C09157=1149.476,8.134,-48.383,179.808,6.183,149.173
C09158=1149.470,8.383,-48.397,179.810,6.184,149.172
C09159=1149.465,8.633,-48.412,179.813,6.186,149.172
C09160=1149.460,8.883,-48.425,179.816,6.186,149.171
C09161=1149.455,9.132,-48.438,179.818,6.187,149.171
C09162=1149.450,9.382,-48.452,179.821,6.187,149.170
C09163=1149.444,9.631,-48.466,179.823,6.188,149.169
C09164=1149.440,9.881,-48.480,179.826,6.189,149.169
C09165=1149.435,10.131,-48.493,179.828,6.190,149.168
C09166=1149.429,10.380,-48.507,179.830,6.191,149.168
C09167=1149.424,10.630,-48.521,179.833,6.191,149.167
C09168=1149.419,10.879,-48.534,179.835,6.192,149.167
C09169=1149.414,11.129,-48.548,179.838,6.193,149.166
C09170=1149.409,11.379,-48.562,179.841,6.194,149.165
C09171=1149.403,11.628,-48.576,179.843,6.195,149.165
C09172=1149.399,11.877,-48.589,179.845,6.196,149.164
C09173=1149.394,12.126,-48.603,179.849,6.197,149.164
C09174=1149.388,12.377,-48.617,179.851,6.198,149.163
C09175=1149.383,12.627,-48.631,179.853,6.198,149.163
C09176=1149.378,12.876,-48.645,179.856,6.199,149.162
C09177=1149.373,13.126,-48.658,179.858,6.201,149.162
C09178=1149.368,13.375,-48.672,179.861,6.201,149.161
C09179=1149.363,13.624,-48.686,179.863,6.202,149.160
C09180=1149.358,13.874,-48.700,179.866,6.202,149.160
C09181=1149.352,14.124,-48.714,179.868,6.203,149.159
C09182=1149.347,14.373,-48.728,179.871,6.204,149.159
C09183=1149.343,14.623,-48.742,179.873,6.205,149.158
C09184=1149.338,14.872,-48.756,179.876,6.206,149.157
C09185=1149.332,15.121,-48.770,179.878,6.206,149.157
C09186=1149.327,15.372,-48.783,179.882,6.208,149.156
C09187=1149.322,15.621,-48.798,179.884,6.208,149.156
C09188=1149.316,15.870,-48.812,179.886,6.209,149.155
C09189=1149.311,16.120,-48.826,179.889,6.210,149.155
C09190=1149.307,16.370,-48.840,179.891,6.211,149.154
C09191=1149.302,16.619,-48.853,179.894,6.212,149.154
C09192=1149.297,16.868,-48.868,179.896,6.213,149.153
C09193=1149.291,17.119,-48.881,179.899,6.213,149.152
C09194=1149.287,17.368,-48.896,179.902,6.215,149.152
C09195=1149.281,17.617,-48.909,179.904,6.215,149.151
C09196=1149.276,17.867,-48.924,179.906,6.216,149.151
C09197=1149.271,18.117,-48.938,179.909,6.218,149.150
C09198=1149.266,18.367,-48.952,179.912,6.218,149.150
C09199=1149.261,18.616,-48.966,179.914,6.219,149.149
C09200=1149.256,18.865,-48.980,179.917,6.219,149.149
C09201=1149.251,19.115,-48.995,179.919,6.221,149.148
C09202=1149.246,19.364,-49.008,179.922,6.221,149.147
C09203=1149.241,19.613,-49.022,179.924,6.222,149.147
C09204=1149.236,19.863,-49.037,179.927,6.223,149.146
C09205=1149.231,20.113,-49.051,179.930,6.224,149.146
C09206=1149.226,20.362,-49.065,179.932,6.225,149.145
C09207=1149.220,20.611,-49.079,179.934,6.226,149.145
C09208=1149.215,20.861,-49.093,179.937,6.227,149.144
C09209=1149.211,21.111,-49.108,179.940,6.228,149.144
C09210=1149.206,21.361,-49.122,179.942,6.229,149.143
C09211=1149.200,21.610,-49.136,179.945,6.229,149.142
C09212=1149.195,21.859,-49.150,179.947,6.231,149.142
C09213=1149.190,22.109,-49.164,179.950,6.231,149.141
C09214=1149.185,22.359,-49.179,179.952,6.232,149.141
C09215=1149.179,22.609,-49.194,179.955,6.233,149.140
C09216=1149.174,22.858,-49.207,179.958,6.234,149.140
C09217=1149.169,23.107,-49.222,179.960,6.235,149.139
C09218=1149.164,23.357,-49.236,179.962,6.235,149.139
C09219=1149.159,23.607,-49.250,179.965,6.237,149.138
C09220=1149.154,23.857,-49.265,179.968,6.237,149.137
C09221=1149.149,24.106,-49.280,179.970,6.238,149.137
C09222=1149.144,24.355,-49.293,179.973,6.239,149.136
C09223=1149.139,24.604,-49.308,179.975,6.240,149.136
C09224=1149.134,24.854,-49.322,179.978,6.241,149.135
C09225=1149.129,25.104,-49.336,179.981,6.242,149.135
C09226=1149.124,25.354,-49.351,179.983,6.243,149.134
C09227=1149.119,25.603,-49.366,179.986,6.244,149.134
C09228=1149.113,25.852,-49.380,179.988,6.245,149.133
C09229=1149.108,26.102,-49.394,179.991,6.246,149.132
C09230=1149.103,26.351,-49.409,179.993,6.247,149.132
C09231=1149.098,26.601,-49.423,179.996,6.247,149.131
C09232=1149.094,26.850,-49.438,179.999,6.249,149.131
C09233=1149.089,27.100,-49.452,-179.999,6.249,149.130
C09234=1149.083,27.369,-49.468,-179.996,6.251,149.130
C09235=1149.077,27.638,-49.483,-179.993,6.251,149.129
C09236=1149.072,27.907,-49.499,-179.991,6.253,149.129
C09237=1149.067,28.175,-49.515,-179.988,6.253,149.128
C09238=1149.061,28.425,-49.529,-179.986,6.254,149.127
C09239=1149.056,28.675,-49.544,-179.982,6.255,149.127
C09240=1149.051,28.924,-49.559,-179.980,6.256,149.126
C09241=1149.046,29.174,-49.573,-179.978,6.257,149.126
C09242=1149.041,29.424,-49.587,-179.975,6.258,149.125
C09243=1149.036,29.673,-49.603,-179.972,6.259,149.125
C09244=1149.031,29.923,-49.617,-179.970,6.260,149.124
C09245=1149.026,30.172,-49.631,-179.967,6.261,149.124
C09246=1149.021,30.421,-49.646,-179.965,6.262,149.123
C09247=1149.016,30.671,-49.661,-179.962,6.263,149.122
C09248=1149.011,30.921,-49.676,-179.959,6.264,149.122
C09249=1149.006,31.170,-49.690,-179.957,6.265,149.121
C09250=1149.001,31.419,-49.704,-179.954,6.266,149.121
C09251=1148.995,31.669,-49.720,-179.952,6.267,149.120
C09252=1148.990,31.918,-49.734,-179.950,6.268,149.120
C09253=1148.986,32.167,-49.749,-179.946,6.269,149.119
C09254=1148.981,32.417,-49.764,-179.944,6.270,149.119
C09255=1148.975,32.667,-49.778,-179.942,6.270,149.118
C09256=1148.970,32.916,-49.793,-179.939,6.272,149.118
C09257=1148.965,33.166,-49.808,-179.936,6.272,149.117
C09258=1148.960,33.415,-49.823,-179.934,6.273,149.116
C09259=1148.955,33.665,-49.838,-179.931,6.275,149.116
C09260=1148.950,33.914,-49.853,-179.929,6.275,149.115
C09261=1148.945,34.164,-49.867,-179.926,6.277,149.115
C09262=1148.940,34.413,-49.882,-179.923,6.277,149.114
C09263=1148.935,34.663,-49.897,-179.921,6.278,149.114
C09264=1148.930,34.912,-49.912,-179.918,6.279,149.113
C09265=1148.925,35.162,-49.927,-179.916,6.280,149.113
C09266=1148.920,35.411,-49.942,-179.913,6.281,149.112
C09267=1148.914,35.661,-49.956,-179.910,6.282,149.111
C09268=1148.910,35.910,-49.971,-179.908,6.283,149.111
C09269=1148.904,36.160,-49.987,-179.905,6.284,149.110
C09270=1148.899,36.409,-50.001,-179.903,6.285,149.110
C09271=1148.895,36.659,-50.016,-179.900,6.286,149.109
C09272=1148.890,36.909,-50.031,-179.897,6.287,149.109
C09273=1148.885,37.158,-50.046,-179.895,6.288,149.108
C09274=1148.880,37.408,-50.062,-179.892,6.289,149.108
C09275=1148.875,37.658,-50.076,-179.890,6.290,149.107
C09276=1148.869,37.907,-50.092,-179.887,6.291,149.106
C09277=1148.864,38.157,-50.106,-179.884,6.292,149.106
C09278=1148.860,38.406,-50.121,-179.882,6.293,149.106
C09279=1148.854,38.655,-50.137,-179.879,6.294,149.105
C09280=1148.849,38.905,-50.151,-179.877,6.295,149.104
C09281=1148.844,39.154,-50.167,-179.874,6.296,149.104
C09282=1148.839,39.403,-50.182,-179.871,6.297,149.103
C09283=1148.834,39.653,-50.197,-179.869,6.298,149.103
C09284=1148.829,39.902,-50.212,-179.866,6.299,149.102
C09285=1148.823,40.152,-50.227,-179.864,6.300,149.102
C09286=1148.819,40.402,-50.242,-179.861,6.301,149.101
C09287=1148.814,40.652,-50.257,-179.858,6.302,149.101
C09288=1148.809,40.901,-50.272,-179.856,6.303,149.100
C09289=1148.804,41.150,-50.288,-179.853,6.305,149.100
C09290=1148.799,41.399,-50.303,-179.851,6.305,149.099
C09291=1148.793,41.649,-50.318,-179.848,6.306,149.098
C09292=1148.789,41.898,-50.333,-179.845,6.308,149.098
C09293=1148.783,42.148,-50.348,-179.843,6.308,149.097
C09294=1148.779,42.398,-50.364,-179.840,6.310,149.097
C09295=1148.774,42.647,-50.379,-179.838,6.310,149.096
C09296=1148.768,42.897,-50.394,-179.835,6.312,149.096
C09297=1148.764,43.146,-50.409,-179.832,6.313,149.095
C09298=1148.758,43.395,-50.425,-179.830,6.313,149.095
C09299=1148.754,43.645,-50.440,-179.827,6.315,149.094
C09300=1148.749,43.895,-50.456,-179.825,6.316,149.094
C09301=1148.743,44.144,-50.471,-179.822,6.317,149.093
C09302=1148.739,44.393,-50.486,-179.819,6.318,149.093
C09303=1148.733,44.643,-50.501,-179.816,6.319,149.092
C09304=1148.728,44.892,-50.516,-179.814,6.320,149.091
C09305=1148.723,45.142,-50.532,-179.811,6.321,149.091
C09306=1148.718,45.392,-50.548,-179.809,6.322,149.090
C09307=1148.714,45.641,-50.563,-179.806,6.323,149.090
C09308=1148.708,45.890,-50.578,-179.803,6.324,149.089
C09309=1148.703,46.140,-50.594,-179.801,6.325,149.089
C09310=1148.698,46.389,-50.609,-179.798,6.326,149.088
C09311=1148.693,46.639,-50.625,-179.796,6.327,149.088
C09312=1148.688,46.888,-50.640,-179.793,6.329,149.087
C09313=1148.683,47.137,-50.655,-179.790,6.329,149.087
C09314=1148.678,47.387,-50.671,-179.788,6.331,149.086
C09315=1148.673,47.637,-50.687,-179.785,6.332,149.086
C09316=1148.668,47.886,-50.702,-179.782,6.333,149.085
C09317=1148.663,48.135,-50.718,-179.780,6.334,149.085
C09318=1148.658,48.385,-50.733,-179.777,6.334,149.084
C09319=1148.654,48.635,-50.748,-179.775,6.336,149.083
C09320=1148.648,48.884,-50.764,-179.772,6.337,149.083
C09321=1148.643,49.133,-50.780,-179.769,6.338,149.082
C09322=1148.637,49.383,-50.795,-179.767,6.339,149.082
C09323=1148.633,49.633,-50.811,-179.764,6.340,149.081
C09324=1148.628,49.882,-50.826,-179.762,6.341,149.081
C09325=1148.623,50.131,-50.842,-179.759,6.343,149.080
C09326=1148.618,50.381,-50.858,-179.756,6.343,149.080
C09327=1148.614,50.630,-50.873,-179.754,6.345,149.079
C09328=1148.608,50.879,-50.889,-179.751,6.346,149.079
C09329=1148.603,51.129,-50.905,-179.748,6.347,149.078
C09330=1148.598,51.379,-50.921,-179.746,6.348,149.078
C09331=1148.593,51.628,-50.936,-179.743,6.349,149.077
C09332=1148.588,51.877,-50.951,-179.741,6.350,149.077
C09333=1148.583,52.127,-50.968,-179.738,6.351,149.076
C09334=1148.578,52.376,-50.983,-179.735,6.352,149.075
C09335=1148.573,52.626,-50.999,-179.732,6.354,149.075
C09336=1148.568,52.876,-51.015,-179.730,6.354,149.074
C09337=1148.563,53.125,-51.030,-179.727,6.356,149.074
C09338=1148.558,53.393,-51.047,-179.725,6.357,149.073
C09339=1148.552,53.662,-51.064,-179.722,6.358,149.073
C09340=1148.547,53.931,-51.081,-179.718,6.359,149.072
C09341=1148.542,54.199,-51.098,-179.716,6.360,149.072
C09342=1148.536,54.449,-51.114,-179.713,6.361,149.071
C09343=1148.531,54.698,-51.130,-179.711,6.362,149.071
C09344=1148.526,54.948,-51.146,-179.708,6.364,149.070
C09345=1148.521,55.197,-51.162,-179.705,6.365,149.069
C09346=1148.517,55.446,-51.178,-179.703,6.366,149.069
C09347=1148.512,55.696,-51.193,-179.700,6.368,149.069
C09348=1148.506,55.945,-51.209,-179.697,6.368,149.068
C09349=1148.502,56.195,-51.226,-179.695,6.370,149.068
C09350=1148.497,56.444,-51.241,-179.692,6.370,149.067
C09351=1148.491,56.693,-51.257,-179.689,6.372,149.066
C09352=1148.487,56.943,-51.274,-179.687,6.373,149.066
C09353=1148.481,57.192,-51.289,-179.684,6.374,149.065
C09354=1148.477,57.442,-51.305,-179.682,6.375,149.065
C09355=1148.471,57.691,-51.321,-179.679,6.376,149.064
C09356=1148.466,57.941,-51.337,-179.676,6.377,149.064
C09357=1148.462,58.190,-51.354,-179.674,6.379,149.063
C09358=1148.456,58.439,-51.369,-179.671,6.379,149.063
C09359=1148.451,58.690,-51.385,-179.668,6.381,149.062
C09360=1148.446,58.938,-51.402,-179.666,6.382,149.062
C09361=1148.442,59.188,-51.417,-179.663,6.383,149.061
C09362=1148.436,59.437,-51.434,-179.660,6.384,149.061
C09363=1148.432,59.687,-51.450,-179.658,6.385,149.060
C09364=1148.427,59.936,-51.466,-179.655,6.387,149.060
C09365=1148.421,60.186,-51.482,-179.652,6.387,149.059
C09366=1148.417,60.435,-51.498,-179.650,6.389,149.059
C09367=1148.411,60.684,-51.514,-179.647,6.390,149.058
C09368=1148.407,60.934,-51.531,-179.644,6.391,149.058
C09369=1148.401,61.183,-51.546,-179.642,6.392,149.057
C09370=1148.397,61.433,-51.563,-179.639,6.393,149.056
C09371=1148.392,61.682,-51.578,-179.637,6.394,149.056
C09372=1148.387,61.932,-51.595,-179.634,6.396,149.056
C09373=1148.382,62.181,-51.611,-179.631,6.397,149.055
C09374=1148.377,62.431,-51.627,-179.629,6.398,149.055
C09375=1148.372,62.679,-51.644,-179.625,6.399,149.054
C09376=1148.367,62.930,-51.660,-179.623,6.400,149.053
C09377=1148.362,63.179,-51.676,-179.621,6.402,149.053
C09378=1148.357,63.429,-51.692,-179.618,6.402,149.052
C09379=1148.352,63.677,-51.709,-179.615,6.404,149.052
C09380=1148.347,63.927,-51.725,-179.612,6.406,149.051
C09381=1148.342,64.176,-51.741,-179.610,6.406,149.051
C09382=1148.337,64.426,-51.758,-179.607,6.408,149.050
C09383=1148.332,64.675,-51.774,-179.605,6.409,149.050
C09384=1148.327,64.925,-51.790,-179.602,6.410,149.049
C09385=1148.322,65.174,-51.807,-179.600,6.411,149.049
C09386=1148.317,65.423,-51.823,-179.597,6.412,149.048
C09387=1148.312,65.673,-51.839,-179.594,6.414,149.048
C09388=1148.307,65.922,-51.856,-179.591,6.415,149.047
C09389=1148.303,66.172,-51.872,-179.589,6.416,149.047
C09390=1148.297,66.421,-51.889,-179.586,6.417,149.046
C09391=1148.292,66.671,-51.905,-179.583,6.418,149.046
C09392=1148.288,66.920,-51.922,-179.581,6.420,149.045
C09393=1148.283,67.169,-51.938,-179.578,6.421,149.045
C09394=1148.278,67.419,-51.955,-179.575,6.422,149.044
C09395=1148.272,67.668,-51.971,-179.573,6.423,149.044
C09396=1148.268,67.918,-51.988,-179.570,6.424,149.043
C09397=1148.263,68.167,-52.004,-179.567,6.426,149.043
C09398=1148.258,68.416,-52.021,-179.565,6.427,149.042
C09399=1148.253,68.666,-52.038,-179.562,6.428,149.042
C09400=1148.247,68.915,-52.054,-179.559,6.429,149.041
C09401=1148.243,69.165,-52.070,-179.557,6.431,149.041
C09402=1148.238,69.414,-52.087,-179.554,6.432,149.040
C09403=1148.233,69.663,-52.104,-179.551,6.433,149.040
C09404=1148.228,69.913,-52.120,-179.549,6.435,149.039
C09405=1148.224,70.162,-52.137,-179.545,6.436,149.039
C09406=1148.218,70.411,-52.154,-179.543,6.437,149.038
C09407=1148.213,70.661,-52.171,-179.540,6.438,149.038
C09408=1148.208,70.910,-52.186,-179.538,6.439,149.037
C09409=1148.203,71.160,-52.204,-179.535,6.441,149.037
C09410=1148.198,71.410,-52.220,-179.532,6.442,149.036
C09411=1148.193,71.658,-52.237,-179.530,6.443,149.036
C09412=1148.188,71.908,-52.254,-179.527,6.444,149.035
C09413=1148.184,72.158,-52.270,-179.524,6.446,149.035
C09414=1148.178,72.406,-52.287,-179.522,6.446,149.034
C09415=1148.173,72.656,-52.304,-179.519,6.448,149.034
C09416=1148.169,72.906,-52.321,-179.517,6.449,149.033
C09417=1148.164,73.155,-52.337,-179.514,6.450,149.032
C09418=1148.158,73.404,-52.354,-179.511,6.452,149.032
C09419=1148.154,73.654,-52.371,-179.509,6.453,149.032
C09420=1148.149,73.904,-52.388,-179.506,6.455,149.031
C09421=1148.144,74.152,-52.405,-179.503,6.456,149.031
C09422=1148.139,74.402,-52.421,-179.501,6.457,149.030
C09423=1148.134,74.652,-52.438,-179.498,6.458,149.030
C09424=1148.130,74.901,-52.455,-179.495,6.460,149.029
C09425=1148.124,75.150,-52.473,-179.492,6.460,149.029
C09426=1148.120,75.399,-52.489,-179.490,6.462,149.028
C09427=1148.114,75.649,-52.507,-179.486,6.463,149.027
C09428=1148.110,75.898,-52.523,-179.484,6.464,149.027
C09429=1148.104,76.147,-52.540,-179.482,6.466,149.027
C09430=1148.100,76.397,-52.557,-179.478,6.467,149.026
C09431=1148.094,76.647,-52.574,-179.476,6.468,149.026
C09432=1148.090,76.896,-52.591,-179.473,6.470,149.025
C09433=1148.084,77.145,-52.608,-179.471,6.471,149.025
C09434=1148.080,77.394,-52.625,-179.468,6.472,149.024
C09435=1148.075,77.644,-52.642,-179.465,6.474,149.024
C09436=1148.070,77.893,-52.659,-179.463,6.475,149.023
C09437=1148.064,78.142,-52.676,-179.460,6.476,149.023
C09438=1148.060,78.392,-52.693,-179.457,6.477,149.022
C09439=1148.055,78.641,-52.711,-179.454,6.479,149.022
C09440=1148.050,78.891,-52.727,-179.452,6.480,149.021
C09441=1148.045,79.140,-52.745,-179.449,6.481,149.021
C09442=1148.040,79.408,-52.762,-179.446,6.483,149.020
C09443=1148.035,79.677,-52.781,-179.443,6.484,149.020
C09444=1148.029,79.945,-52.800,-179.440,6.486,149.019
C09445=1148.024,80.213,-52.818,-179.437,6.487,149.018
C09446=1148.019,80.463,-52.835,-179.435,6.488,149.018
C09447=1148.014,80.713,-52.853,-179.432,6.490,149.018
C09448=1148.010,80.962,-52.870,-179.430,6.491,149.017
C09449=1148.004,81.211,-52.887,-179.427,6.492,149.016
C09450=1147.999,81.460,-52.904,-179.424,6.494,149.016
C09451=1147.994,81.709,-52.922,-179.421,6.495,149.016
C09452=1147.989,81.959,-52.939,-179.419,6.496,149.015
C09453=1147.985,82.209,-52.955,-179.416,6.498,149.015
C09454=1147.980,82.458,-52.973,-179.413,6.499,149.014
C09455=1147.975,82.708,-52.991,-179.411,6.501,149.014
C09456=1147.970,82.956,-53.008,-179.408,6.501,149.013
C09457=1147.965,83.206,-53.025,-179.405,6.503,149.013
C09458=1147.959,83.455,-53.042,-179.402,6.505,149.012
C09459=1147.955,83.704,-53.060,-179.400,6.506,149.012
C09460=1147.950,83.954,-53.077,-179.397,6.507,149.011
C09461=1147.945,84.203,-53.095,-179.394,6.509,149.011
C09462=1147.941,84.453,-53.112,-179.392,6.510,149.010
C09463=1147.936,84.702,-53.130,-179.389,6.511,149.010
C09464=1147.930,84.952,-53.147,-179.386,6.512,149.009
C09465=1147.926,85.201,-53.164,-179.384,6.514,149.009
C09466=1147.920,85.450,-53.181,-179.381,6.516,149.008
C09467=1147.916,85.699,-53.199,-179.378,6.516,149.008
C09468=1147.910,85.949,-53.216,-179.375,6.518,149.007
C09469=1147.906,86.198,-53.234,-179.373,6.520,149.007
C09470=1147.901,86.447,-53.251,-179.371,6.520,149.006
C09471=1147.896,86.697,-53.269,-179.367,6.522,149.006
C09472=1147.891,86.946,-53.286,-179.365,6.523,149.005
C09473=1147.887,87.195,-53.304,-179.362,6.525,149.005
C09474=1147.882,87.444,-53.322,-179.360,6.526,149.005
C09475=1147.877,87.694,-53.339,-179.357,6.527,149.004
C09476=1147.872,87.943,-53.357,-179.354,6.529,149.003
C09477=1147.866,88.193,-53.374,-179.351,6.531,149.003
C09478=1147.862,88.442,-53.391,-179.349,6.532,149.003
C09479=1147.857,88.691,-53.409,-179.346,6.533,149.002
C09480=1147.852,88.941,-53.427,-179.343,6.535,149.002
C09481=1147.847,89.190,-53.445,-179.340,6.536,149.001
C09482=1147.842,89.439,-53.463,-179.338,6.537,149.001
C09483=1147.837,89.689,-53.480,-179.335,6.538,149.000
C09484=1147.833,89.938,-53.497,-179.332,6.540,149.000
C09485=1147.828,90.187,-53.515,-179.329,6.542,148.999
C09486=1147.823,90.437,-53.533,-179.327,6.543,148.999
C09487=1147.818,90.686,-53.551,-179.324,6.544,148.998
C09488=1147.813,90.935,-53.569,-179.321,6.546,148.998
C09489=1147.808,91.184,-53.587,-179.319,6.547,148.997
C09490=1147.803,91.434,-53.604,-179.316,6.549,148.997
C09491=1147.798,91.683,-53.622,-179.313,6.549,148.996
C09492=1147.793,91.933,-53.640,-179.310,6.551,148.996
C09493=1147.788,92.182,-53.658,-179.308,6.553,148.995
C09494=1147.784,92.431,-53.674,-179.305,6.554,148.995
C09495=1147.779,92.680,-53.692,-179.302,6.555,148.994
C09496=1147.774,92.930,-53.710,-179.300,6.557,148.994
C09497=1147.769,93.179,-53.728,-179.297,6.558,148.993
C09498=1147.764,93.428,-53.746,-179.294,6.560,148.993
C09499=1147.759,93.677,-53.764,-179.291,6.562,148.993
C09500=1147.754,93.928,-53.782,-179.289,6.562,148.992
C09501=1147.749,94.177,-53.800,-179.286,6.564,148.992
C09502=1147.745,94.426,-53.818,-179.283,6.566,148.991
C09503=1147.740,94.675,-53.836,-179.281,6.567,148.991
C09504=1147.735,94.924,-53.854,-179.277,6.569,148.990
C09505=1147.730,95.174,-53.872,-179.275,6.569,148.990
C09506=1147.725,95.423,-53.890,-179.273,6.571,148.989
C09507=1147.720,95.672,-53.908,-179.270,6.573,148.989
C09508=1147.715,95.921,-53.926,-179.267,6.575,148.988
C09509=1147.710,96.170,-53.944,-179.264,6.576,148.988
C09510=1147.706,96.420,-53.962,-179.262,6.577,148.987
C09511=1147.701,96.669,-53.980,-179.259,6.578,148.987
C09512=1147.696,96.918,-53.998,-179.256,6.580,148.987
C09513=1147.691,97.168,-54.016,-179.253,6.582,148.986
C09514=1147.686,97.417,-54.035,-179.250,6.583,148.985
C09515=1147.681,97.666,-54.053,-179.248,6.584,148.985
C09516=1147.676,97.915,-54.071,-179.245,6.586,148.985
C09517=1147.671,98.165,-54.089,-179.243,6.587,148.984
C09518=1147.666,98.415,-54.107,-179.239,6.589,148.984
C09519=1147.662,98.664,-54.125,-179.237,6.590,148.983
C09520=1147.657,98.913,-54.143,-179.234,6.592,148.983
C09521=1147.652,99.162,-54.161,-179.232,6.593,148.982
C09522=1147.647,99.411,-54.179,-179.229,6.595,148.982
C09523=1147.642,99.661,-54.198,-179.226,6.596,148.982
C09524=1147.637,99.911,-54.216,-179.223,6.598,148.981
C09525=1147.632,100.160,-54.234,-179.220,6.599,148.980
C09526=1147.627,100.409,-54.252,-179.218,6.601,148.980
C09527=1147.622,100.657,-54.270,-179.216,6.602,148.980
C09528=1147.618,100.907,-54.289,-179.213,6.603,148.979
C09529=1147.612,101.157,-54.307,-179.210,6.605,148.979
C09530=1147.608,101.406,-54.325,-179.207,6.607,148.978
C09531=1147.603,101.655,-54.343,-179.204,6.608,148.978
C09532=1147.598,101.905,-54.362,-179.201,6.610,148.977
C09533=1147.594,102.154,-54.380,-179.199,6.612,148.977
C09534=1147.588,102.403,-54.399,-179.196,6.612,148.976
C09535=1147.583,102.652,-54.417,-179.193,6.614,148.976
C09536=1147.578,102.901,-54.435,-179.191,6.615,148.975
C09537=1147.574,103.151,-54.454,-179.188,6.617,148.975
C09538=1147.569,103.400,-54.472,-179.185,6.619,148.975
C09539=1147.564,103.649,-54.490,-179.182,6.621,148.974
C09540=1147.559,103.899,-54.509,-179.179,6.622,148.974
C09541=1147.555,104.148,-54.528,-179.177,6.623,148.973
C09542=1147.549,104.397,-54.546,-179.174,6.624,148.973
C09543=1147.544,104.647,-54.564,-179.172,6.626,148.972
C09544=1147.540,104.896,-54.583,-179.169,6.628,148.972
C09545=1147.535,105.145,-54.601,-179.166,6.629,148.971
C09546=1147.529,105.414,-54.621,-179.163,6.631,148.971
C09547=1147.524,105.682,-54.641,-179.160,6.632,148.970
C09548=1147.519,105.950,-54.662,-179.158,6.634,148.970
C09549=1147.514,106.219,-54.681,-179.154,6.635,148.969
C09550=1147.509,106.468,-54.700,-179.152,6.637,148.969
C09551=1147.504,106.717,-54.718,-179.149,6.639,148.969
C09552=1147.500,106.967,-54.737,-179.146,6.641,148.968
C09553=1147.494,107.215,-54.756,-179.143,6.642,148.968
C09554=1147.490,107.465,-54.774,-179.140,6.644,148.967
C09555=1147.485,107.714,-54.792,-179.137,6.645,148.967
C09556=1147.480,107.963,-54.812,-179.135,6.647,148.966
C09557=1147.475,108.213,-54.830,-179.133,6.648,148.966
C09558=1147.470,108.462,-54.849,-179.130,6.650,148.965
C09559=1147.465,108.711,-54.867,-179.127,6.651,148.965
C09560=1147.461,108.961,-54.886,-179.124,6.653,148.964
C09561=1147.456,109.210,-54.905,-179.121,6.654,148.964
C09562=1147.451,109.459,-54.923,-179.118,6.656,148.964
C09563=1147.446,109.709,-54.942,-179.116,6.658,148.963
C09564=1147.441,109.957,-54.961,-179.113,6.659,148.963
C09565=1147.436,110.206,-54.980,-179.110,6.661,148.962
C09566=1147.432,110.456,-54.999,-179.108,6.663,148.962
C09567=1147.426,110.705,-55.018,-179.104,6.664,148.961
C09568=1147.422,110.955,-55.036,-179.102,6.665,148.961
C09569=1147.418,111.203,-55.055,-179.100,6.667,148.961
C09570=1147.412,111.453,-55.074,-179.097,6.668,148.960
C09571=1147.408,111.702,-55.093,-179.094,6.670,148.960
C09572=1147.403,111.951,-55.112,-179.091,6.672,148.959
C09573=1147.397,112.201,-55.131,-179.089,6.673,148.959
C09574=1147.393,112.450,-55.150,-179.086,6.675,148.959
C09575=1147.388,112.699,-55.169,-179.083,6.676,148.958
C09576=1147.383,112.948,-55.187,-179.080,6.678,148.957
C09577=1147.378,113.197,-55.207,-179.077,6.680,148.957
C09578=1147.374,113.447,-55.226,-179.075,6.681,148.957
C09579=1147.368,113.696,-55.244,-179.072,6.683,148.956
C09580=1147.364,113.945,-55.263,-179.069,6.685,148.956
C09581=1147.359,114.194,-55.283,-179.066,6.687,148.955
C09582=1147.355,114.443,-55.302,-179.064,6.687,148.955
C09583=1147.349,114.693,-55.320,-179.061,6.689,148.954
C09584=1147.344,114.943,-55.340,-179.058,6.690,148.954
C09585=1147.340,115.191,-55.359,-179.056,6.692,148.954
C09586=1147.335,115.441,-55.378,-179.053,6.694,148.953
C09587=1147.330,115.690,-55.396,-179.050,6.696,148.953
C09588=1147.325,115.939,-55.416,-179.047,6.697,148.952
C09589=1147.320,116.188,-55.435,-179.045,6.699,148.952
C09590=1147.316,116.438,-55.454,-179.042,6.701,148.952
C09591=1147.311,116.686,-55.473,-179.039,6.702,148.951
C09592=1147.306,116.937,-55.492,-179.036,6.704,148.951
C09593=1147.301,117.185,-55.511,-179.033,6.705,148.950
C09594=1147.296,117.435,-55.531,-179.031,6.707,148.950
C09595=1147.291,117.684,-55.550,-179.028,6.709,148.949
C09596=1147.287,117.933,-55.569,-179.025,6.710,148.949
C09597=1147.282,118.182,-55.588,-179.022,6.712,148.949
C09598=1147.277,118.431,-55.608,-179.020,6.714,148.948
C09599=1147.272,118.680,-55.627,-179.017,6.716,148.948
C09600=1147.268,118.929,-55.646,-179.014,6.717,148.947
C09601=1147.263,119.179,-55.666,-179.011,6.719,148.947
C09602=1147.257,119.428,-55.685,-179.009,6.721,148.947
C09603=1147.253,119.677,-55.704,-179.006,6.722,148.946
C09604=1147.248,119.927,-55.723,-179.003,6.724,148.945
C09605=1147.243,120.176,-55.743,-179.000,6.725,148.945
C09606=1147.238,120.425,-55.762,-178.997,6.727,148.945
C09607=1147.234,120.674,-55.781,-178.995,6.729,148.944
C09608=1147.229,120.923,-55.801,-178.992,6.730,148.944
C09609=1147.224,121.172,-55.821,-178.989,6.732,148.943
C09610=1147.219,121.422,-55.840,-178.987,6.734,148.943
C09611=1147.215,121.670,-55.859,-178.984,6.736,148.943
C09612=1147.210,121.920,-55.879,-178.981,6.737,148.942
C09613=1147.205,122.169,-55.898,-178.978,6.739,148.942
C09614=1147.200,122.418,-55.918,-178.976,6.741,148.941
C09615=1147.195,122.668,-55.937,-178.973,6.742,148.941
C09616=1147.190,122.917,-55.957,-178.970,6.744,148.940
C09617=1147.186,123.166,-55.976,-178.967,6.745,148.940
C09618=1147.181,123.415,-55.995,-178.964,6.747,148.940
C09619=1147.176,123.665,-56.015,-178.962,6.749,148.939
C09620=1147.171,123.913,-56.035,-178.959,6.751,148.939
C09621=1147.166,124.163,-56.055,-178.956,6.752,148.938
C09622=1147.162,124.412,-56.074,-178.953,6.754,148.938
C09623=1147.156,124.661,-56.094,-178.951,6.756,148.938
C09624=1147.152,124.911,-56.113,-178.948,6.757,148.937
C09625=1147.148,125.159,-56.133,-178.945,6.759,148.937
C09626=1147.143,125.408,-56.152,-178.943,6.761,148.936
C09627=1147.138,125.658,-56.172,-178.940,6.762,148.936
C09628=1147.133,125.907,-56.192,-178.937,6.764,148.936
C09629=1147.128,126.156,-56.212,-178.934,6.766,148.935
C09630=1147.123,126.405,-56.231,-178.932,6.768,148.935
C09631=1147.119,126.655,-56.251,-178.929,6.769,148.934
C09632=1147.114,126.904,-56.271,-178.926,6.771,148.934
C09633=1147.109,127.153,-56.291,-178.923,6.773,148.934
C09634=1147.104,127.402,-56.310,-178.921,6.774,148.933
C09635=1147.099,127.652,-56.330,-178.918,6.776,148.933
C09636=1147.094,127.900,-56.350,-178.915,6.777,148.932
C09637=1147.089,128.150,-56.370,-178.912,6.779,148.932
C09638=1147.085,128.399,-56.389,-178.909,6.781,148.931
C09639=1147.080,128.648,-56.410,-178.907,6.783,148.931
C09640=1147.075,128.897,-56.429,-178.904,6.784,148.931
C09641=1147.070,129.147,-56.449,-178.901,6.787,148.930
C09642=1147.066,129.396,-56.469,-178.898,6.788,148.930
C09643=1147.061,129.645,-56.489,-178.895,6.790,148.929
C09644=1147.056,129.893,-56.509,-178.893,6.792,148.929
C09645=1147.051,130.143,-56.528,-178.890,6.794,148.929
C09646=1147.047,130.392,-56.549,-178.887,6.795,148.928
C09647=1147.042,130.641,-56.568,-178.884,6.797,148.928
C09648=1147.038,130.890,-56.589,-178.882,6.799,148.928
C09649=1147.032,131.139,-56.608,-178.879,6.800,148.927
C09650=1147.027,131.408,-56.630,-178.876,6.802,148.927
C09651=1147.022,131.676,-56.651,-178.873,6.805,148.926
C09652=1147.017,131.945,-56.672,-178.870,6.806,148.926
C09653=1147.011,132.214,-56.694,-178.867,6.808,148.926
C09654=1147.007,132.463,-56.715,-178.864,6.809,148.925
C09655=1147.002,132.712,-56.734,-178.862,6.811,148.925
C09656=1146.998,132.961,-56.755,-178.858,6.814,148.924
C09657=1146.993,133.210,-56.775,-178.856,6.815,148.924
C09658=1146.987,133.459,-56.795,-178.853,6.817,148.923
C09659=1146.983,133.708,-56.815,-178.850,6.819,148.923
C09660=1146.978,133.958,-56.835,-178.848,6.821,148.923
C09661=1146.974,134.207,-56.855,-178.845,6.822,148.922
C09662=1146.969,134.456,-56.876,-178.842,6.824,148.922
C09663=1146.965,134.705,-56.895,-178.840,6.826,148.922
C09664=1146.959,134.955,-56.916,-178.837,6.828,148.921
C09665=1146.954,135.204,-56.936,-178.834,6.829,148.921
C09666=1146.950,135.453,-56.956,-178.831,6.832,148.920
C09667=1146.945,135.701,-56.976,-178.828,6.834,148.920
C09668=1146.940,135.951,-56.997,-178.826,6.835,148.920
C09669=1146.935,136.200,-57.017,-178.823,6.837,148.919
C09670=1146.931,136.449,-57.037,-178.820,6.839,148.919
C09671=1146.926,136.698,-57.058,-178.817,6.840,148.919
C09672=1146.921,136.948,-57.078,-178.815,6.842,148.918
C09673=1146.916,137.197,-57.098,-178.812,6.844,148.918
C09674=1146.912,137.446,-57.119,-178.809,6.845,148.917
C09675=1146.908,137.695,-57.139,-178.806,6.848,148.917
C09676=1146.902,137.943,-57.160,-178.803,6.850,148.917
C09677=1146.897,138.193,-57.179,-178.801,6.851,148.916
C09678=1146.893,138.442,-57.200,-178.798,6.853,148.916
C09679=1146.887,138.691,-57.221,-178.795,6.855,148.915
C09680=1146.883,138.940,-57.241,-178.792,6.857,148.915
C09681=1146.879,139.189,-57.261,-178.790,6.858,148.915
C09682=1146.873,139.439,-57.282,-178.787,6.860,148.914
C09683=1146.869,139.688,-57.302,-178.784,6.863,148.914
C09684=1146.864,139.937,-57.322,-178.781,6.864,148.913
C09685=1146.859,140.186,-57.343,-178.778,6.866,148.913
C09686=1146.855,140.435,-57.364,-178.776,6.868,148.913
C09687=1146.850,140.684,-57.384,-178.773,6.869,148.912
C09688=1146.845,140.933,-57.405,-178.770,6.871,148.912
C09689=1146.841,141.182,-57.425,-178.767,6.873,148.912
C09690=1146.836,141.431,-57.446,-178.764,6.875,148.911
C09691=1146.831,141.680,-57.467,-178.761,6.877,148.911
C09692=1146.826,141.929,-57.487,-178.759,6.879,148.911
C09693=1146.821,142.179,-57.508,-178.756,6.881,148.910
C09694=1146.817,142.428,-57.528,-178.754,6.883,148.910
C09695=1146.812,142.677,-57.549,-178.751,6.884,148.909
C09696=1146.807,142.926,-57.570,-178.748,6.887,148.909
C09697=1146.803,143.175,-57.590,-178.745,6.888,148.909
C09698=1146.798,143.424,-57.611,-178.742,6.890,148.908
C09699=1146.793,143.673,-57.631,-178.740,6.892,148.908
C09700=1146.788,143.922,-57.652,-178.737,6.894,148.907
C09701=1146.784,144.172,-57.673,-178.734,6.895,148.907
C09702=1146.779,144.421,-57.694,-178.731,6.898,148.907
C09703=1146.775,144.670,-57.715,-178.728,6.900,148.906
C09704=1146.769,144.919,-57.735,-178.725,6.901,148.906
C09705=1146.765,145.168,-57.756,-178.723,6.903,148.906
C09706=1146.760,145.417,-57.778,-178.720,6.905,148.905
C09707=1146.756,145.666,-57.798,-178.718,6.907,148.905
C09708=1146.750,145.915,-57.819,-178.714,6.909,148.905
C09709=1146.746,146.164,-57.839,-178.712,6.911,148.904
C09710=1146.741,146.413,-57.860,-178.709,6.913,148.904
C09711=1146.736,146.663,-57.881,-178.706,6.914,148.903
C09712=1146.732,146.912,-57.903,-178.704,6.916,148.903
C09713=1146.727,147.161,-57.924,-178.700,6.919,148.903
C09714=1146.723,147.410,-57.944,-178.698,6.920,148.902
C09715=1146.717,147.659,-57.965,-178.695,6.922,148.902
C09716=1146.713,147.908,-57.985,-178.692,6.924,148.902
C09717=1146.708,148.157,-58.007,-178.690,6.926,148.901
C09718=1146.703,148.406,-58.028,-178.687,6.928,148.901
C09719=1146.698,148.655,-58.048,-178.684,6.930,148.901
C09720=1146.694,148.904,-58.070,-178.681,6.932,148.900
C09721=1146.689,149.154,-58.091,-178.679,6.934,148.900
C09722=1146.685,149.403,-58.112,-178.676,6.935,148.900
C09723=1146.680,149.651,-58.133,-178.673,6.938,148.899
C09724=1146.675,149.900,-58.154,-178.670,6.940,148.899
C09725=1146.670,150.149,-58.175,-178.667,6.941,148.898
C09726=1146.666,150.399,-58.197,-178.665,6.943,148.898
C09727=1146.661,150.648,-58.218,-178.662,6.945,148.898
C09728=1146.656,150.897,-58.238,-178.659,6.948,148.897
C09729=1146.651,151.146,-58.260,-178.656,6.949,148.897
C09730=1146.646,151.395,-58.281,-178.653,6.951,148.897
C09731=1146.642,151.644,-58.303,-178.651,6.953,148.896
C09732=1146.637,151.893,-58.323,-178.647,6.955,148.896
C09733=1146.632,152.142,-58.344,-178.645,6.957,148.896
C09734=1146.627,152.391,-58.366,-178.642,6.959,148.895
C09735=1146.623,152.640,-58.386,-178.640,6.961,148.895
C09736=1146.619,152.889,-58.408,-178.636,6.963,148.895
C09737=1146.614,153.139,-58.429,-178.634,6.965,148.894
C09738=1146.609,153.387,-58.451,-178.631,6.967,148.894
C09739=1146.604,153.636,-58.472,-178.628,6.968,148.894
C09740=1146.600,153.885,-58.493,-178.625,6.971,148.893
C09741=1146.595,154.135,-58.514,-178.623,6.973,148.893
C09742=1146.590,154.383,-58.536,-178.620,6.975,148.893
C09743=1146.585,154.632,-58.558,-178.617,6.977,148.892
C09744=1146.580,154.882,-58.579,-178.614,6.979,148.892
C09745=1146.576,155.130,-58.600,-178.611,6.981,148.891
C09746=1146.571,155.380,-58.621,-178.609,6.982,148.891
C09747=1146.567,155.629,-58.643,-178.606,6.985,148.891
C09748=1146.562,155.878,-58.664,-178.603,6.987,148.891
C09749=1146.557,156.127,-58.686,-178.600,6.989,148.890
C09750=1146.552,156.375,-58.707,-178.598,6.991,148.890
C09751=1146.547,156.625,-58.729,-178.595,6.992,148.889
C09752=1146.543,156.874,-58.750,-178.592,6.995,148.889
C09753=1146.538,157.122,-58.772,-178.590,6.997,148.889
C09754=1146.533,157.392,-58.795,-178.587,6.999,148.889
C09755=1146.528,157.661,-58.818,-178.584,7.001,148.888
C09756=1146.523,157.930,-58.842,-178.580,7.004,148.888
C09757=1146.518,158.199,-58.864,-178.578,7.005,148.887
C09758=1146.513,158.447,-58.886,-178.575,7.007,148.887
C09759=1146.509,158.697,-58.908,-178.572,7.010,148.887
C09760=1146.504,158.946,-58.929,-178.569,7.011,148.886
C09761=1146.500,159.195,-58.951,-178.566,7.013,148.886
C09762=1146.495,159.444,-58.973,-178.564,7.015,148.886
C09763=1146.490,159.692,-58.995,-178.561,7.018,148.885
C09764=1146.485,159.942,-59.016,-178.558,7.019,148.885
C09765=1146.481,160.191,-59.038,-178.555,7.021,148.885
C09766=1146.476,160.440,-59.059,-178.552,7.024,148.884
C09767=1146.471,160.689,-59.081,-178.550,7.026,148.884
C09768=1146.467,160.938,-59.103,-178.547,7.027,148.884
C09769=1146.462,161.187,-59.125,-178.544,7.030,148.883
C09770=1146.457,161.436,-59.147,-178.541,7.032,148.883
C09771=1146.453,161.684,-59.168,-178.538,7.033,148.883
C09772=1146.448,161.934,-59.190,-178.536,7.036,148.883
C09773=1146.443,162.183,-59.211,-178.533,7.038,148.882
C09774=1146.439,162.432,-59.234,-178.530,7.040,148.882
C09775=1146.434,162.681,-59.255,-178.527,7.042,148.881
C09776=1146.429,162.931,-59.278,-178.524,7.044,148.881
C09777=1146.424,163.179,-59.300,-178.522,7.046,148.881
C09778=1146.420,163.428,-59.322,-178.519,7.048,148.881
C09779=1146.415,163.677,-59.343,-178.516,7.050,148.880
C09780=1146.410,163.926,-59.365,-178.513,7.052,148.880
C09781=1146.406,164.175,-59.387,-178.511,7.054,148.880
C09782=1146.401,164.424,-59.409,-178.508,7.057,148.879
C09783=1146.397,164.673,-59.431,-178.505,7.058,148.879
C09784=1146.392,164.922,-59.452,-178.502,7.060,148.879
C09785=1146.387,165.171,-59.475,-178.499,7.063,148.878
C09786=1146.382,165.420,-59.497,-178.497,7.065,148.878
C09787=1146.378,165.669,-59.519,-178.494,7.067,148.878
C09788=1146.373,165.917,-59.541,-178.491,7.069,148.877
C09789=1146.369,166.167,-59.563,-178.488,7.071,148.877
C09790=1146.364,166.415,-59.585,-178.486,7.073,148.877
C09791=1146.359,166.665,-59.608,-178.483,7.075,148.876
C09792=1146.354,166.914,-59.629,-178.480,7.077,148.876
C09793=1146.350,167.163,-59.651,-178.478,7.079,148.876
C09794=1146.345,167.412,-59.673,-178.474,7.082,148.876
C09795=1146.340,167.661,-59.696,-178.472,7.084,148.875
C09796=1146.335,167.909,-59.718,-178.469,7.085,148.875
C09797=1146.331,168.159,-59.740,-178.466,7.088,148.875
C09798=1146.327,168.408,-59.762,-178.463,7.090,148.874
C09799=1146.321,168.657,-59.784,-178.460,7.092,148.874
C09800=1146.317,168.906,-59.807,-178.457,7.094,148.874
C09801=1146.312,169.154,-59.829,-178.455,7.096,148.873
C09802=1146.308,169.404,-59.851,-178.452,7.099,148.873
C09803=1146.302,169.653,-59.873,-178.449,7.100,148.873
C09804=1146.299,169.901,-59.896,-178.446,7.102,148.872
C09805=1146.294,170.151,-59.918,-178.444,7.105,148.872
C09806=1146.289,170.400,-59.940,-178.441,7.107,148.872
C09807=1146.285,170.648,-59.963,-178.438,7.109,148.872
C09808=1146.280,170.897,-59.985,-178.435,7.111,148.871
C09809=1146.275,171.147,-60.007,-178.433,7.113,148.871
C09810=1146.271,171.395,-60.030,-178.429,7.116,148.871
C09811=1146.266,171.644,-60.052,-178.427,7.117,148.870
C09812=1146.261,171.893,-60.075,-178.425,7.120,148.870
C09813=1146.256,172.142,-60.097,-178.421,7.122,148.870
C09814=1146.251,172.391,-60.119,-178.419,7.124,148.869
C09815=1146.247,172.640,-60.142,-178.416,7.127,148.869
C09816=1146.243,172.889,-60.164,-178.413,7.128,148.869
C09817=1146.238,173.138,-60.187,-178.410,7.130,148.869
C09818=1146.234,173.387,-60.209,-178.407,7.133,148.868
C09819=1146.228,173.635,-60.232,-178.405,7.135,148.868
C09820=1146.224,173.885,-60.254,-178.402,7.137,148.868
C09821=1146.220,174.133,-60.277,-178.399,7.139,148.867
C09822=1146.214,174.382,-60.299,-178.397,7.141,148.867
C09823=1146.211,174.631,-60.322,-178.393,7.144,148.867
C09824=1146.206,174.881,-60.345,-178.391,7.145,148.866
C09825=1146.201,175.129,-60.367,-178.388,7.148,148.866
C09826=1146.196,175.378,-60.390,-178.385,7.150,148.866
C09827=1146.192,175.627,-60.413,-178.382,7.152,148.866
C09828=1146.186,175.876,-60.435,-178.380,7.155,148.865
C09829=1146.182,176.125,-60.458,-178.377,7.156,148.865
C09830=1146.178,176.374,-60.481,-178.374,7.159,148.865
C09831=1146.173,176.623,-60.503,-178.371,7.161,148.865
C09832=1146.168,176.872,-60.526,-178.368,7.164,148.864
C09833=1146.164,177.121,-60.548,-178.365,7.165,148.864
C09834=1146.159,177.370,-60.571,-178.363,7.167,148.864
C09835=1146.155,177.619,-60.594,-178.360,7.170,148.863
C09836=1146.150,177.868,-60.616,-178.357,7.172,148.863
C09837=1146.145,178.117,-60.640,-178.354,7.175,148.863
C09838=1146.141,178.365,-60.663,-178.352,7.176,148.863
C09839=1146.136,178.614,-60.686,-178.348,7.179,148.862
C09840=1146.131,178.863,-60.708,-178.346,7.181,148.862
C09841=1146.127,179.112,-60.731,-178.344,7.183,148.862
C09842=1146.122,179.361,-60.754,-178.340,7.185,148.861
C09843=1146.118,179.610,-60.777,-178.338,7.187,148.861
C09844=1146.112,179.859,-60.799,-178.335,7.190,148.861
C09845=1146.108,180.107,-60.822,-178.333,7.192,148.861
C09846=1146.104,180.356,-60.846,-178.329,7.195,148.860
C09847=1146.099,180.606,-60.869,-178.327,7.196,148.860
C09848=1146.095,180.854,-60.892,-178.324,7.199,148.860
C09849=1146.090,181.104,-60.914,-178.321,7.201,148.860
C09850=1146.085,181.352,-60.937,-178.318,7.203,148.859
C09851=1146.081,181.601,-60.960,-178.316,7.206,148.859
C09852=1146.076,181.850,-60.983,-178.313,7.207,148.859
C09853=1146.071,182.099,-61.007,-178.310,7.210,148.858
C09854=1146.067,182.348,-61.030,-178.307,7.212,148.858
C09855=1146.063,182.597,-61.053,-178.304,7.214,148.858
C09856=1146.057,182.845,-61.076,-178.302,7.217,148.858
C09857=1146.053,183.094,-61.099,-178.299,7.219,148.857
C09858=1146.048,183.364,-61.124,-178.295,7.222,148.857
C09859=1146.043,183.633,-61.149,-178.293,7.224,148.857
C09860=1146.038,183.904,-61.174,-178.290,7.226,148.857
C09861=1146.033,184.174,-61.199,-178.286,7.229,148.856
C09862=1146.029,184.422,-61.222,-178.284,7.231,148.856
C09863=1146.024,184.671,-61.245,-178.281,7.233,148.856
C09864=1146.019,184.920,-61.268,-178.278,7.235,148.855
C09865=1146.014,185.169,-61.292,-178.275,7.238,148.855
C09866=1146.010,185.417,-61.316,-178.273,7.240,148.855
C09867=1146.006,185.666,-61.338,-178.270,7.243,148.855
C09868=1146.001,185.915,-61.362,-178.267,7.244,148.854
C09869=1145.996,186.164,-61.385,-178.264,7.247,148.854
C09870=1145.992,186.413,-61.409,-178.262,7.249,148.854
C09871=1145.987,186.662,-61.432,-178.259,7.252,148.854
C09872=1145.982,186.911,-61.455,-178.256,7.254,148.853
C09873=1145.978,187.160,-61.478,-178.253,7.256,148.853
C09874=1145.974,187.409,-61.501,-178.250,7.258,148.853
C09875=1145.969,187.657,-61.525,-178.248,7.261,148.853
C09876=1145.965,187.906,-61.549,-178.245,7.263,148.852
C09877=1145.959,188.155,-61.572,-178.242,7.266,148.852
C09878=1145.955,188.404,-61.595,-178.239,7.267,148.852
C09879=1145.950,188.653,-61.619,-178.237,7.270,148.852
C09880=1145.945,188.901,-61.643,-178.234,7.272,148.851
C09881=1145.941,189.150,-61.666,-178.231,7.275,148.851
C09882=1145.936,189.399,-61.689,-178.228,7.277,148.851
C09883=1145.931,189.648,-61.713,-178.225,7.279,148.851
C09884=1145.927,189.897,-61.737,-178.222,7.282,148.850
C09885=1145.922,190.146,-61.760,-178.220,7.284,148.850
C09886=1145.918,190.395,-61.783,-178.217,7.287,148.850
C09887=1145.913,190.644,-61.807,-178.214,7.288,148.850
C09888=1145.908,190.892,-61.831,-178.211,7.291,148.849
C09889=1145.904,191.141,-61.854,-178.209,7.293,148.849
C09890=1145.899,191.390,-61.878,-178.206,7.296,148.849
C09891=1145.895,191.639,-61.902,-178.203,7.298,148.849
C09892=1145.890,191.888,-61.925,-178.200,7.301,148.849
C09893=1145.886,192.136,-61.949,-178.198,7.302,148.848
C09894=1145.881,192.386,-61.973,-178.194,7.305,148.848
C09895=1145.877,192.635,-61.996,-178.192,7.307,148.848
C09896=1145.872,192.883,-62.020,-178.189,7.310,148.847
C09897=1145.868,193.132,-62.044,-178.186,7.313,148.847
C09898=1145.863,193.381,-62.068,-178.183,7.314,148.847
C09899=1145.859,193.630,-62.091,-178.180,7.317,148.847
C09900=1145.854,193.878,-62.115,-178.178,7.319,148.846
C09901=1145.849,194.127,-62.139,-178.175,7.322,148.846
C09902=1145.845,194.375,-62.163,-178.172,7.324,148.846
C09903=1145.840,194.625,-62.187,-178.169,7.326,148.846
C09904=1145.835,194.873,-62.211,-178.166,7.329,148.846
C09905=1145.831,195.122,-62.234,-178.164,7.331,148.845
C09906=1145.827,195.371,-62.258,-178.161,7.334,148.845
C09907=1145.822,195.620,-62.282,-178.159,7.336,148.845
C09908=1145.818,195.869,-62.306,-178.155,7.338,148.845
C09909=1145.813,196.118,-62.329,-178.153,7.340,148.844
C09910=1145.808,196.367,-62.354,-178.150,7.343,148.844
C09911=1145.803,196.615,-62.378,-178.147,7.346,148.844
C09912=1145.799,196.864,-62.401,-178.144,7.348,148.844
C09913=1145.794,197.112,-62.425,-178.141,7.351,148.844
C09914=1145.791,197.362,-62.450,-178.139,7.352,148.843
C09915=1145.785,197.611,-62.474,-178.136,7.355,148.843
C09916=1145.781,197.859,-62.498,-178.134,7.357,148.843
C09917=1145.776,198.108,-62.522,-178.130,7.360,148.843
C09918=1145.772,198.357,-62.545,-178.128,7.363,148.842
C09919=1145.767,198.605,-62.570,-178.125,7.364,148.842
C09920=1145.763,198.855,-62.594,-178.122,7.367,148.842
C09921=1145.758,199.104,-62.618,-178.119,7.369,148.842
C09922=1145.754,199.352,-62.642,-178.117,7.372,148.842
C09923=1145.748,199.601,-62.666,-178.113,7.375,148.841
C09924=1145.744,199.849,-62.691,-178.111,7.377,148.841
C09925=1145.740,200.098,-62.715,-178.108,7.379,148.841
C09926=1145.735,200.348,-62.739,-178.106,7.381,148.841
C09927=1145.730,200.596,-62.763,-178.102,7.384,148.840
C09928=1145.726,200.844,-62.787,-178.100,7.387,148.840
C09929=1145.722,201.094,-62.812,-178.097,7.389,148.840
C09930=1145.717,201.342,-62.836,-178.094,7.391,148.840
C09931=1145.713,201.591,-62.860,-178.091,7.394,148.840
C09932=1145.707,201.840,-62.884,-178.089,7.396,148.839
C09933=1145.704,202.089,-62.909,-178.086,7.399,148.839
C09934=1145.699,202.338,-62.933,-178.083,7.401,148.839
C09935=1145.694,202.586,-62.957,-178.080,7.404,148.839
C09936=1145.690,202.835,-62.982,-178.078,7.407,148.839
C09937=1145.686,203.084,-63.006,-178.075,7.408,148.838
C09938=1145.681,203.333,-63.031,-178.072,7.411,148.838
C09939=1145.676,203.581,-63.055,-178.069,7.414,148.838
C09940=1145.672,203.830,-63.080,-178.067,7.416,148.838
C09941=1145.667,204.079,-63.104,-178.063,7.418,148.837
C09942=1145.662,204.328,-63.128,-178.061,7.421,148.837
C09943=1145.658,204.577,-63.153,-178.058,7.423,148.837
C09944=1145.654,204.825,-63.177,-178.055,7.426,148.837
C09945=1145.649,205.074,-63.202,-178.053,7.428,148.837
C09946=1145.645,205.322,-63.226,-178.050,7.431,148.836
C09947=1145.640,205.572,-63.251,-178.047,7.434,148.836
C09948=1145.636,205.820,-63.275,-178.045,7.436,148.836
C09949=1145.630,206.069,-63.300,-178.041,7.438,148.836
C09950=1145.627,206.318,-63.324,-178.038,7.441,148.836
C09951=1145.622,206.566,-63.349,-178.036,7.443,148.835
C09952=1145.617,206.815,-63.374,-178.033,7.446,148.835
C09953=1145.613,207.064,-63.398,-178.030,7.449,148.835
C09954=1145.608,207.313,-63.423,-178.027,7.451,148.835
C09955=1145.604,207.562,-63.448,-178.025,7.453,148.835
C09956=1145.599,207.810,-63.472,-178.022,7.456,148.835
C09957=1145.594,208.059,-63.496,-178.019,7.458,148.834
C09958=1145.590,208.308,-63.522,-178.016,7.461,148.834
C09959=1145.585,208.556,-63.547,-178.013,7.464,148.834
C09960=1145.581,208.805,-63.571,-178.011,7.466,148.834
C09961=1145.576,209.054,-63.596,-178.008,7.469,148.834
C09962=1145.571,209.324,-63.623,-178.005,7.471,148.833
C09963=1145.566,209.595,-63.650,-178.002,7.474,148.833
C09964=1145.561,209.865,-63.676,-177.999,7.477,148.833
C09965=1145.557,210.136,-63.703,-177.996,7.480,148.833
C09966=1145.552,210.384,-63.729,-177.993,7.482,148.832
C09967=1145.547,210.634,-63.754,-177.990,7.484,148.832
C09968=1145.543,210.882,-63.778,-177.988,7.487,148.832
C09969=1145.539,211.131,-63.804,-177.984,7.490,148.832
C09970=1145.534,211.380,-63.828,-177.982,7.493,148.832
C09971=1145.530,211.629,-63.853,-177.979,7.495,148.832
C09972=1145.525,211.877,-63.878,-177.976,7.497,148.831
C09973=1145.521,212.126,-63.903,-177.973,7.500,148.831
C09974=1145.516,212.374,-63.928,-177.971,7.502,148.831
C09975=1145.512,212.624,-63.953,-177.968,7.505,148.831
C09976=1145.507,212.872,-63.978,-177.965,7.508,148.831
C09977=1145.503,213.121,-64.003,-177.963,7.510,148.831
C09978=1145.498,213.369,-64.028,-177.960,7.512,148.830
C09979=1145.494,213.618,-64.053,-177.957,7.515,148.830
C09980=1145.489,213.867,-64.078,-177.954,7.518,148.830
C09981=1145.485,214.116,-64.104,-177.952,7.520,148.830
C09982=1145.480,214.364,-64.128,-177.948,7.523,148.830
C09983=1145.476,214.613,-64.154,-177.946,7.526,148.830
C09984=1145.471,214.861,-64.179,-177.943,7.528,148.829
C09985=1145.467,215.111,-64.204,-177.940,7.530,148.829
C09986=1145.462,215.359,-64.229,-177.937,7.533,148.829
C09987=1145.458,215.608,-64.254,-177.935,7.536,148.829
C09988=1145.453,215.856,-64.279,-177.932,7.538,148.829
C09989=1145.449,216.105,-64.304,-177.929,7.541,148.829
C09990=1145.444,216.353,-64.330,-177.926,7.544,148.828
C09991=1145.440,216.602,-64.355,-177.924,7.547,148.828
C09992=1145.435,216.852,-64.380,-177.921,7.549,148.828
C09993=1145.430,217.100,-64.406,-177.918,7.551,148.828
C09994=1145.427,217.348,-64.431,-177.915,7.554,148.828
C09995=1145.422,217.597,-64.456,-177.912,7.557,148.827
C09996=1145.417,217.846,-64.481,-177.910,7.559,148.827
//INST
///DATE 2021/06/15 17:27
///ATTR SC,RW,RJ
////FRAME ROBOT
///GROUP1 RB1
NOP
MOVL C00000 V=800.0 PL=0
MOVL C00001 V=800.0 PL=0
MOVL C00002 V=800.0 PL=0
MOVL C00003 V=800.0 PL=0
MOVL C00004 V=800.0 PL=0
MOVL C00005 V=800.0 PL=0
MOVL C00006 V=800.0 PL=0
MOVL C00007 V=800.0 PL=0
MOVL C00008 V=800.0 PL=0
MOVL C00009 V=800.0 PL=0
MOVL C00010 V=800.0 PL=0
MOVL C00011 V=800.0 PL=0
MOVL C00012 V=800.0 PL=0
MOVL C00013 V=800.0 PL=0
MOVL C00014 V=800.0 PL=0
MOVL C00015 V=800.0 PL=0
MOVL C00016 V=800.0 PL=0
MOVL C00017 V=800.0 PL=0
MOVL C00018 V=800.0 PL=0
MOVL C00019 V=800.0 PL=0
MOVL C00020 V=800.0 PL=0
MOVL C00021 V=800.0 PL=0
MOVL C00022 V=800.0 PL=0
MOVL C00023 V=800.0 PL=0
MOVL C00024 V=800.0 PL=0
MOVL C00025 V=800.0 PL=0
MOVL C00026 V=800.0 PL=0
MOVL C00027 V=800.0 PL=0
MOVL C00028 V=800.0 PL=0
MOVL C00029 V=800.0 PL=0
MOVL C00030 V=800.0 PL=0
MOVL C00031 V=800.0 PL=0
MOVL C00032 V=800.0 PL=0
MOVL C00033 V=800.0 PL=0
MOVL C00034 V=800.0 PL=0
MOVL C00035 V=800.0 PL=0
MOVL C00036 V=800.0 PL=0
MOVL C00037 V=800.0 PL=0
MOVL C00038 V=800.0 PL=0
MOVL C00039 V=800.0 PL=0
MOVL C00040 V=800.0 PL=0
MOVL C00041 V=800.0 PL=0
MOVL C00042 V=800.0 PL=0
MOVL C00043 V=800.0 PL=0
MOVL C00044 V=800.0 PL=0
MOVL C00045 V=800.0 PL=0
MOVL C00046 V=800.0 PL=0
MOVL C00047 V=800.0 PL=0
MOVL C00048 V=800.0 PL=0
MOVL C00049 V=800.0 PL=0
MOVL C00050 V=800.0 PL=0
MOVL C00051 V=800.0 PL=0
MOVL C00052 V=800.0 PL=0
MOVL C00053 V=800.0 PL=0
MOVL C00054 V=800.0 PL=0
MOVL C00055 V=800.0 PL=0
MOVL C00056 V=800.0 PL=0
MOVL C00057 V=800.0 PL=0
MOVL C00058 V=800.0 PL=0
MOVL C00059 V=800.0 PL=0
MOVL C00060 V=800.0 PL=0
MOVL C00061 V=800.0 PL=0
MOVL C00062 V=800.0 PL=0
MOVL C00063 V=800.0 PL=0
MOVL C00064 V=800.0 PL=0
MOVL C00065 V=800.0 PL=0
MOVL C00066 V=800.0 PL=0
MOVL C00067 V=800.0 PL=0
MOVL C00068 V=800.0 PL=0
MOVL C00069 V=800.0 PL=0
MOVL C00070 V=800.0 PL=0
MOVL C00071 V=800.0 PL=0
MOVL C00072 V=800.0 PL=0
MOVL C00073 V=800.0 PL=0
MOVL C00074 V=800.0 PL=0
MOVL C00075 V=800.0 PL=0
MOVL C00076 V=800.0 PL=0
MOVL C00077 V=800.0 PL=0
MOVL C00078 V=800.0 PL=0
MOVL C00079 V=800.0 PL=0
MOVL C00080 V=800.0 PL=0
MOVL C00081 V=800.0 PL=0
MOVL C00082 V=800.0 PL=0
MOVL C00083 V=800.0 PL=0
MOVL C00084 V=800.0 PL=0
MOVL C00085 V=800.0 PL=0
MOVL C00086 V=800.0 PL=0
MOVL C00087 V=800.0 PL=0
MOVL C00088 V=800.0 PL=0
MOVL C00089 V=800.0 PL=0
MOVL C00090 V=800.0 PL=0
MOVL C00091 V=800.0 PL=0
MOVL C00092 V=800.0 PL=0
MOVL C00093 V=800.0 PL=0
MOVL C00094 V=800.0 PL=0
MOVL C00095 V=800.0 PL=0
MOVL C00096 V=800.0 PL=0
MOVL C00097 V=800.0 PL=0
MOVL C00098 V=800.0 PL=0
MOVL C00099 V=800.0 PL=0
MOVL C00100 V=800.0 PL=0
MOVL C00101 V=800.0 PL=0
MOVL C00102 V=800.0 PL=0
MOVL C00103 V=800.0 PL=0
MOVL C00104 V=800.0 PL=0
MOVL C00105 V=800.0 PL=0
MOVL C00106 V=800.0 PL=0
MOVL C00107 V=800.0 PL=0
MOVL C00108 V=800.0 PL=0
MOVL C00109 V=800.0 PL=0
MOVL C00110 V=800.0 PL=0
MOVL C00111 V=800.0 PL=0
MOVL C00112 V=800.0 PL=0
MOVL C00113 V=800.0 PL=0
MOVL C00114 V=800.0 PL=0
MOVL C00115 V=800.0 PL=0
MOVL C00116 V=800.0 PL=0
MOVL C00117 V=800.0 PL=0
MOVL C00118 V=800.0 PL=0
MOVL C00119 V=800.0 PL=0
MOVL C00120 V=800.0 PL=0
MOVL C00121 V=800.0 PL=0
MOVL C00122 V=800.0 PL=0
MOVL C00123 V=800.0 PL=0
MOVL C00124 V=800.0 PL=0
MOVL C00125 V=800.0 PL=0
MOVL C00126 V=800.0 PL=0
MOVL C00127 V=800.0 PL=0
MOVL C00128 V=800.0 PL=0
MOVL C00129 V=800.0 PL=0
MOVL C00130 V=800.0 PL=0
MOVL C00131 V=800.0 PL=0
MOVL C00132 V=800.0 PL=0
MOVL C00133 V=800.0 PL=0
MOVL C00134 V=800.0 PL=0
MOVL C00135 V=800.0 PL=0
MOVL C00136 V=800.0 PL=0
MOVL C00137 V=800.0 PL=0
MOVL C00138 V=800.0 PL=0
MOVL C00139 V=800.0 PL=0
MOVL C00140 V=800.0 PL=0
MOVL C00141 V=800.0 PL=0
MOVL C00142 V=800.0 PL=0
MOVL C00143 V=800.0 PL=0
MOVL C00144 V=800.0 PL=0
MOVL C00145 V=800.0 PL=0
MOVL C00146 V=800.0 PL=0
MOVL C00147 V=800.0 PL=0
MOVL C00148 V=800.0 PL=0
MOVL C00149 V=800.0 PL=0
MOVL C00150 V=800.0 PL=0
MOVL C00151 V=800.0 PL=0
MOVL C00152 V=800.0 PL=0
MOVL C00153 V=800.0 PL=0
MOVL C00154 V=800.0 PL=0
MOVL C00155 V=800.0 PL=0
MOVL C00156 V=800.0 PL=0
MOVL C00157 V=800.0 PL=0
MOVL C00158 V=800.0 PL=0
MOVL C00159 V=800.0 PL=0
MOVL C00160 V=800.0 PL=0
MOVL C00161 V=800.0 PL=0
MOVL C00162 V=800.0 PL=0
MOVL C00163 V=800.0 PL=0
MOVL C00164 V=800.0 PL=0
MOVL C00165 V=800.0 PL=0
MOVL C00166 V=800.0 PL=0
MOVL C00167 V=800.0 PL=0
MOVL C00168 V=800.0 PL=0
MOVL C00169 V=800.0 PL=0
MOVL C00170 V=800.0 PL=0
MOVL C00171 V=800.0 PL=0
MOVL C00172 V=800.0 PL=0
MOVL C00173 V=800.0 PL=0
MOVL C00174 V=800.0 PL=0
MOVL C00175 V=800.0 PL=0
MOVL C00176 V=800.0 PL=0
MOVL C00177 V=800.0 PL=0
MOVL C00178 V=800.0 PL=0
MOVL C00179 V=800.0 PL=0
MOVL C00180 V=800.0 PL=0
MOVL C00181 V=800.0 PL=0
MOVL C00182 V=800.0 PL=0
MOVL C00183 V=800.0 PL=0
MOVL C00184 V=800.0 PL=0
MOVL C00185 V=800.0 PL=0
MOVL C00186 V=800.0 PL=0
MOVL C00187 V=800.0 PL=0
MOVL C00188 V=800.0 PL=0
MOVL C00189 V=800.0 PL=0
MOVL C00190 V=800.0 PL=0
MOVL C00191 V=800.0 PL=0
MOVL C00192 V=800.0 PL=0
MOVL C00193 V=800.0 PL=0
MOVL C00194 V=800.0 PL=0
MOVL C00195 V=800.0 PL=0
MOVL C00196 V=800.0 PL=0
MOVL C00197 V=800.0 PL=0
MOVL C00198 V=800.0 PL=0
MOVL C00199 V=800.0 PL=0
MOVL C00200 V=800.0 PL=0
MOVL C00201 V=800.0 PL=0
MOVL C00202 V=800.0 PL=0
MOVL C00203 V=800.0 PL=0
MOVL C00204 V=800.0 PL=0
MOVL C00205 V=800.0 PL=0
MOVL C00206 V=800.0 PL=0
MOVL C00207 V=800.0 PL=0
MOVL C00208 V=800.0 PL=0
MOVL C00209 V=800.0 PL=0
MOVL C00210 V=800.0 PL=0
MOVL C00211 V=800.0 PL=0
MOVL C00212 V=800.0 PL=0
MOVL C00213 V=800.0 PL=0
MOVL C00214 V=800.0 PL=0
MOVL C00215 V=800.0 PL=0
MOVL C00216 V=800.0 PL=0
MOVL C00217 V=800.0 PL=0
MOVL C00218 V=800.0 PL=0
MOVL C00219 V=800.0 PL=0
MOVL C00220 V=800.0 PL=0
MOVL C00221 V=800.0 PL=0
MOVL C00222 V=800.0 PL=0
MOVL C00223 V=800.0 PL=0
MOVL C00224 V=800.0 PL=0
MOVL C00225 V=800.0 PL=0
MOVL C00226 V=800.0 PL=0
MOVL C00227 V=800.0 PL=0
MOVL C00228 V=800.0 PL=0
MOVL C00229 V=800.0 PL=0
MOVL C00230 V=800.0 PL=0
MOVL C00231 V=800.0 PL=0
MOVL C00232 V=800.0 PL=0
MOVL C00233 V=800.0 PL=0
MOVL C00234 V=800.0 PL=0
MOVL C00235 V=800.0 PL=0
MOVL C00236 V=800.0 PL=0
MOVL C00237 V=800.0 PL=0
MOVL C00238 V=800.0 PL=0
MOVL C00239 V=800.0 PL=0
MOVL C00240 V=800.0 PL=0
MOVL C00241 V=800.0 PL=0
MOVL C00242 V=800.0 PL=0
MOVL C00243 V=800.0 PL=0
MOVL C00244 V=800.0 PL=0
MOVL C00245 V=800.0 PL=0
MOVL C00246 V=800.0 PL=0
MOVL C00247 V=800.0 PL=0
MOVL C00248 V=800.0 PL=0
MOVL C00249 V=800.0 PL=0
MOVL C00250 V=800.0 PL=0
MOVL C00251 V=800.0 PL=0
MOVL C00252 V=800.0 PL=0
MOVL C00253 V=800.0 PL=0
MOVL C00254 V=800.0 PL=0
MOVL C00255 V=800.0 PL=0
MOVL C00256 V=800.0 PL=0
MOVL C00257 V=800.0 PL=0
MOVL C00258 V=800.0 PL=0
MOVL C00259 V=800.0 PL=0
MOVL C00260 V=800.0 PL=0
MOVL C00261 V=800.0 PL=0
MOVL C00262 V=800.0 PL=0
MOVL C00263 V=800.0 PL=0
MOVL C00264 V=800.0 PL=0
MOVL C00265 V=800.0 PL=0
MOVL C00266 V=800.0 PL=0
MOVL C00267 V=800.0 PL=0
MOVL C00268 V=800.0 PL=0
MOVL C00269 V=800.0 PL=0
MOVL C00270 V=800.0 PL=0
MOVL C00271 V=800.0 PL=0
MOVL C00272 V=800.0 PL=0
MOVL C00273 V=800.0 PL=0
MOVL C00274 V=800.0 PL=0
MOVL C00275 V=800.0 PL=0
MOVL C00276 V=800.0 PL=0
MOVL C00277 V=800.0 PL=0
MOVL C00278 V=800.0 PL=0
MOVL C00279 V=800.0 PL=0
MOVL C00280 V=800.0 PL=0
MOVL C00281 V=800.0 PL=0
MOVL C00282 V=800.0 PL=0
MOVL C00283 V=800.0 PL=0
MOVL C00284 V=800.0 PL=0
MOVL C00285 V=800.0 PL=0
MOVL C00286 V=800.0 PL=0
MOVL C00287 V=800.0 PL=0
MOVL C00288 V=800.0 PL=0
MOVL C00289 V=800.0 PL=0
MOVL C00290 V=800.0 PL=0
MOVL C00291 V=800.0 PL=0
MOVL C00292 V=800.0 PL=0
MOVL C00293 V=800.0 PL=0
MOVL C00294 V=800.0 PL=0
MOVL C00295 V=800.0 PL=0
MOVL C00296 V=800.0 PL=0
MOVL C00297 V=800.0 PL=0
MOVL C00298 V=800.0 PL=0
MOVL C00299 V=800.0 PL=0
MOVL C00300 V=800.0 PL=0
MOVL C00301 V=800.0 PL=0
MOVL C00302 V=800.0 PL=0
MOVL C00303 V=800.0 PL=0
MOVL C00304 V=800.0 PL=0
MOVL C00305 V=800.0 PL=0
MOVL C00306 V=800.0 PL=0
MOVL C00307 V=800.0 PL=0
MOVL C00308 V=800.0 PL=0
MOVL C00309 V=800.0 PL=0
MOVL C00310 V=800.0 PL=0
MOVL C00311 V=800.0 PL=0
MOVL C00312 V=800.0 PL=0
MOVL C00313 V=800.0 PL=0
MOVL C00314 V=800.0 PL=0
MOVL C00315 V=800.0 PL=0
MOVL C00316 V=800.0 PL=0
MOVL C00317 V=800.0 PL=0
MOVL C00318 V=800.0 PL=0
MOVL C00319 V=800.0 PL=0
MOVL C00320 V=800.0 PL=0
MOVL C00321 V=800.0 PL=0
MOVL C00322 V=800.0 PL=0
MOVL C00323 V=800.0 PL=0
MOVL C00324 V=800.0 PL=0
MOVL C00325 V=800.0 PL=0
MOVL C00326 V=800.0 PL=0
MOVL C00327 V=800.0 PL=0
MOVL C00328 V=800.0 PL=0
MOVL C00329 V=800.0 PL=0
MOVL C00330 V=800.0 PL=0
MOVL C00331 V=800.0 PL=0
MOVL C00332 V=800.0 PL=0
MOVL C00333 V=800.0 PL=0
MOVL C00334 V=800.0 PL=0
MOVL C00335 V=800.0 PL=0
MOVL C00336 V=800.0 PL=0
MOVL C00337 V=800.0 PL=0
MOVL C00338 V=800.0 PL=0
MOVL C00339 V=800.0 PL=0
MOVL C00340 V=800.0 PL=0
MOVL C00341 V=800.0 PL=0
MOVL C00342 V=800.0 PL=0
MOVL C00343 V=800.0 PL=0
MOVL C00344 V=800.0 PL=0
MOVL C00345 V=800.0 PL=0
MOVL C00346 V=800.0 PL=0
MOVL C00347 V=800.0 PL=0
MOVL C00348 V=800.0 PL=0
MOVL C00349 V=800.0 PL=0
MOVL C00350 V=800.0 PL=0
MOVL C00351 V=800.0 PL=0
MOVL C00352 V=800.0 PL=0
MOVL C00353 V=800.0 PL=0
MOVL C00354 V=800.0 PL=0
MOVL C00355 V=800.0 PL=0
MOVL C00356 V=800.0 PL=0
MOVL C00357 V=800.0 PL=0
MOVL C00358 V=800.0 PL=0
MOVL C00359 V=800.0 PL=0
MOVL C00360 V=800.0 PL=0
MOVL C00361 V=800.0 PL=0
MOVL C00362 V=800.0 PL=0
MOVL C00363 V=800.0 PL=0
MOVL C00364 V=800.0 PL=0
MOVL C00365 V=800.0 PL=0
MOVL C00366 V=800.0 PL=0
MOVL C00367 V=800.0 PL=0
MOVL C00368 V=800.0 PL=0
MOVL C00369 V=800.0 PL=0
MOVL C00370 V=800.0 PL=0
MOVL C00371 V=800.0 PL=0
MOVL C00372 V=800.0 PL=0
MOVL C00373 V=800.0 PL=0
MOVL C00374 V=800.0 PL=0
MOVL C00375 V=800.0 PL=0
MOVL C00376 V=800.0 PL=0
MOVL C00377 V=800.0 PL=0
MOVL C00378 V=800.0 PL=0
MOVL C00379 V=800.0 PL=0
MOVL C00380 V=800.0 PL=0
MOVL C00381 V=800.0 PL=0
MOVL C00382 V=800.0 PL=0
MOVL C00383 V=800.0 PL=0
MOVL C00384 V=800.0 PL=0
MOVL C00385 V=800.0 PL=0
MOVL C00386 V=800.0 PL=0
MOVL C00387 V=800.0 PL=0
MOVL C00388 V=800.0 PL=0
MOVL C00389 V=800.0 PL=0
MOVL C00390 V=800.0 PL=0
MOVL C00391 V=800.0 PL=0
MOVL C00392 V=800.0 PL=0
MOVL C00393 V=800.0 PL=0
MOVL C00394 V=800.0 PL=0
MOVL C00395 V=800.0 PL=0
MOVL C00396 V=800.0 PL=0
MOVL C00397 V=800.0 PL=0
MOVL C00398 V=800.0 PL=0
MOVL C00399 V=800.0 PL=0
MOVL C00400 V=800.0 PL=0
MOVL C00401 V=800.0 PL=0
MOVL C00402 V=800.0 PL=0
MOVL C00403 V=800.0 PL=0
MOVL C00404 V=800.0 PL=0
MOVL C00405 V=800.0 PL=0
MOVL C00406 V=800.0 PL=0
MOVL C00407 V=800.0 PL=0
MOVL C00408 V=800.0 PL=0
MOVL C00409 V=800.0 PL=0
MOVL C00410 V=800.0 PL=0
MOVL C00411 V=800.0 PL=0
MOVL C00412 V=800.0 PL=0
MOVL C00413 V=800.0 PL=0
MOVL C00414 V=800.0 PL=0
MOVL C00415 V=800.0 PL=0
MOVL C00416 V=800.0 PL=0
MOVL C00417 V=800.0 PL=0
MOVL C00418 V=800.0 PL=0
MOVL C00419 V=800.0 PL=0
MOVL C00420 V=800.0 PL=0
MOVL C00421 V=800.0 PL=0
MOVL C00422 V=800.0 PL=0
MOVL C00423 V=800.0 PL=0
MOVL C00424 V=800.0 PL=0
MOVL C00425 V=800.0 PL=0
MOVL C00426 V=800.0 PL=0
MOVL C00427 V=800.0 PL=0
MOVL C00428 V=800.0 PL=0
MOVL C00429 V=800.0 PL=0
MOVL C00430 V=800.0 PL=0
MOVL C00431 V=800.0 PL=0
MOVL C00432 V=800.0 PL=0
MOVL C00433 V=800.0 PL=0
MOVL C00434 V=800.0 PL=0
MOVL C00435 V=800.0 PL=0
MOVL C00436 V=800.0 PL=0
MOVL C00437 V=800.0 PL=0
MOVL C00438 V=800.0 PL=0
MOVL C00439 V=800.0 PL=0
MOVL C00440 V=800.0 PL=0
MOVL C00441 V=800.0 PL=0
MOVL C00442 V=800.0 PL=0
MOVL C00443 V=800.0 PL=0
MOVL C00444 V=800.0 PL=0
MOVL C00445 V=800.0 PL=0
MOVL C00446 V=800.0 PL=0
MOVL C00447 V=800.0 PL=0
MOVL C00448 V=800.0 PL=0
MOVL C00449 V=800.0 PL=0
MOVL C00450 V=800.0 PL=0
MOVL C00451 V=800.0 PL=0
MOVL C00452 V=800.0 PL=0
MOVL C00453 V=800.0 PL=0
MOVL C00454 V=800.0 PL=0
MOVL C00455 V=800.0 PL=0
MOVL C00456 V=800.0 PL=0
MOVL C00457 V=800.0 PL=0
MOVL C00458 V=800.0 PL=0
MOVL C00459 V=800.0 PL=0
MOVL C00460 V=800.0 PL=0
MOVL C00461 V=800.0 PL=0
MOVL C00462 V=800.0 PL=0
MOVL C00463 V=800.0 PL=0
MOVL C00464 V=800.0 PL=0
MOVL C00465 V=800.0 PL=0
MOVL C00466 V=800.0 PL=0
MOVL C00467 V=800.0 PL=0
MOVL C00468 V=800.0 PL=0
MOVL C00469 V=800.0 PL=0
MOVL C00470 V=800.0 PL=0
MOVL C00471 V=800.0 PL=0
MOVL C00472 V=800.0 PL=0
MOVL C00473 V=800.0 PL=0
MOVL C00474 V=800.0 PL=0
MOVL C00475 V=800.0 PL=0
MOVL C00476 V=800.0 PL=0
MOVL C00477 V=800.0 PL=0
MOVL C00478 V=800.0 PL=0
MOVL C00479 V=800.0 PL=0
MOVL C00480 V=800.0 PL=0
MOVL C00481 V=800.0 PL=0
MOVL C00482 V=800.0 PL=0
MOVL C00483 V=800.0 PL=0
MOVL C00484 V=800.0 PL=0
MOVL C00485 V=800.0 PL=0
MOVL C00486 V=800.0 PL=0
MOVL C00487 V=800.0 PL=0
MOVL C00488 V=800.0 PL=0
MOVL C00489 V=800.0 PL=0
MOVL C00490 V=800.0 PL=0
MOVL C00491 V=800.0 PL=0
MOVL C00492 V=800.0 PL=0
MOVL C00493 V=800.0 PL=0
MOVL C00494 V=800.0 PL=0
MOVL C00495 V=800.0 PL=0
MOVL C00496 V=800.0 PL=0
MOVL C00497 V=800.0 PL=0
MOVL C00498 V=800.0 PL=0
MOVL C00499 V=800.0 PL=0
MOVL C00500 V=800.0 PL=0
MOVL C00501 V=800.0 PL=0
MOVL C00502 V=800.0 PL=0
MOVL C00503 V=800.0 PL=0
MOVL C00504 V=800.0 PL=0
MOVL C00505 V=800.0 PL=0
MOVL C00506 V=800.0 PL=0
MOVL C00507 V=800.0 PL=0
MOVL C00508 V=800.0 PL=0
MOVL C00509 V=800.0 PL=0
MOVL C00510 V=800.0 PL=0
MOVL C00511 V=800.0 PL=0
MOVL C00512 V=800.0 PL=0
MOVL C00513 V=800.0 PL=0
MOVL C00514 V=800.0 PL=0
MOVL C00515 V=800.0 PL=0
MOVL C00516 V=800.0 PL=0
MOVL C00517 V=800.0 PL=0
MOVL C00518 V=800.0 PL=0
MOVL C00519 V=800.0 PL=0
MOVL C00520 V=800.0 PL=0
MOVL C00521 V=800.0 PL=0
MOVL C00522 V=800.0 PL=0
MOVL C00523 V=800.0 PL=0
MOVL C00524 V=800.0 PL=0
MOVL C00525 V=800.0 PL=0
MOVL C00526 V=800.0 PL=0
MOVL C00527 V=800.0 PL=0
MOVL C00528 V=800.0 PL=0
MOVL C00529 V=800.0 PL=0
MOVL C00530 V=800.0 PL=0
MOVL C00531 V=800.0 PL=0
MOVL C00532 V=800.0 PL=0
MOVL C00533 V=800.0 PL=0
MOVL C00534 V=800.0 PL=0
MOVL C00535 V=800.0 PL=0
MOVL C00536 V=800.0 PL=0
MOVL C00537 V=800.0 PL=0
MOVL C00538 V=800.0 PL=0
MOVL C00539 V=800.0 PL=0
MOVL C00540 V=800.0 PL=0
MOVL C00541 V=800.0 PL=0
MOVL C00542 V=800.0 PL=0
MOVL C00543 V=800.0 PL=0
MOVL C00544 V=800.0 PL=0
MOVL C00545 V=800.0 PL=0
MOVL C00546 V=800.0 PL=0
MOVL C00547 V=800.0 PL=0
MOVL C00548 V=800.0 PL=0
MOVL C00549 V=800.0 PL=0
MOVL C00550 V=800.0 PL=0
MOVL C00551 V=800.0 PL=0
MOVL C00552 V=800.0 PL=0
MOVL C00553 V=800.0 PL=0
MOVL C00554 V=800.0 PL=0
MOVL C00555 V=800.0 PL=0
MOVL C00556 V=800.0 PL=0
MOVL C00557 V=800.0 PL=0
MOVL C00558 V=800.0 PL=0
MOVL C00559 V=800.0 PL=0
MOVL C00560 V=800.0 PL=0
MOVL C00561 V=800.0 PL=0
MOVL C00562 V=800.0 PL=0
MOVL C00563 V=800.0 PL=0
MOVL C00564 V=800.0 PL=0
MOVL C00565 V=800.0 PL=0
MOVL C00566 V=800.0 PL=0
MOVL C00567 V=800.0 PL=0
MOVL C00568 V=800.0 PL=0
MOVL C00569 V=800.0 PL=0
MOVL C00570 V=800.0 PL=0
MOVL C00571 V=800.0 PL=0
MOVL C00572 V=800.0 PL=0
MOVL C00573 V=800.0 PL=0
MOVL C00574 V=800.0 PL=0
MOVL C00575 V=800.0 PL=0
MOVL C00576 V=800.0 PL=0
MOVL C00577 V=800.0 PL=0
MOVL C00578 V=800.0 PL=0
MOVL C00579 V=800.0 PL=0
MOVL C00580 V=800.0 PL=0
MOVL C00581 V=800.0 PL=0
MOVL C00582 V=800.0 PL=0
MOVL C00583 V=800.0 PL=0
MOVL C00584 V=800.0 PL=0
MOVL C00585 V=800.0 PL=0
MOVL C00586 V=800.0 PL=0
MOVL C00587 V=800.0 PL=0
MOVL C00588 V=800.0 PL=0
MOVL C00589 V=800.0 PL=0
MOVL C00590 V=800.0 PL=0
MOVL C00591 V=800.0 PL=0
MOVL C00592 V=800.0 PL=0
MOVL C00593 V=800.0 PL=0
MOVL C00594 V=800.0 PL=0
MOVL C00595 V=800.0 PL=0
MOVL C00596 V=800.0 PL=0
MOVL C00597 V=800.0 PL=0
MOVL C00598 V=800.0 PL=0
MOVL C00599 V=800.0 PL=0
MOVL C00600 V=800.0 PL=0
MOVL C00601 V=800.0 PL=0
MOVL C00602 V=800.0 PL=0
MOVL C00603 V=800.0 PL=0
MOVL C00604 V=800.0 PL=0
MOVL C00605 V=800.0 PL=0
MOVL C00606 V=800.0 PL=0
MOVL C00607 V=800.0 PL=0
MOVL C00608 V=800.0 PL=0
MOVL C00609 V=800.0 PL=0
MOVL C00610 V=800.0 PL=0
MOVL C00611 V=800.0 PL=0
MOVL C00612 V=800.0 PL=0
MOVL C00613 V=800.0 PL=0
MOVL C00614 V=800.0 PL=0
MOVL C00615 V=800.0 PL=0
MOVL C00616 V=800.0 PL=0
MOVL C00617 V=800.0 PL=0
MOVL C00618 V=800.0 PL=0
MOVL C00619 V=800.0 PL=0
MOVL C00620 V=800.0 PL=0
MOVL C00621 V=800.0 PL=0
MOVL C00622 V=800.0 PL=0
MOVL C00623 V=800.0 PL=0
MOVL C00624 V=800.0 PL=0
MOVL C00625 V=800.0 PL=0
MOVL C00626 V=800.0 PL=0
MOVL C00627 V=800.0 PL=0
MOVL C00628 V=800.0 PL=0
MOVL C00629 V=800.0 PL=0
MOVL C00630 V=800.0 PL=0
MOVL C00631 V=800.0 PL=0
MOVL C00632 V=800.0 PL=0
MOVL C00633 V=800.0 PL=0
MOVL C00634 V=800.0 PL=0
MOVL C00635 V=800.0 PL=0
MOVL C00636 V=800.0 PL=0
MOVL C00637 V=800.0 PL=0
MOVL C00638 V=800.0 PL=0
MOVL C00639 V=800.0 PL=0
MOVL C00640 V=800.0 PL=0
MOVL C00641 V=800.0 PL=0
MOVL C00642 V=800.0 PL=0
MOVL C00643 V=800.0 PL=0
MOVL C00644 V=800.0 PL=0
MOVL C00645 V=800.0 PL=0
MOVL C00646 V=800.0 PL=0
MOVL C00647 V=800.0 PL=0
MOVL C00648 V=800.0 PL=0
MOVL C00649 V=800.0 PL=0
MOVL C00650 V=800.0 PL=0
MOVL C00651 V=800.0 PL=0
MOVL C00652 V=800.0 PL=0
MOVL C00653 V=800.0 PL=0
MOVL C00654 V=800.0 PL=0
MOVL C00655 V=800.0 PL=0
MOVL C00656 V=800.0 PL=0
MOVL C00657 V=800.0 PL=0
MOVL C00658 V=800.0 PL=0
MOVL C00659 V=800.0 PL=0
MOVL C00660 V=800.0 PL=0
MOVL C00661 V=800.0 PL=0
MOVL C00662 V=800.0 PL=0
MOVL C00663 V=800.0 PL=0
MOVL C00664 V=800.0 PL=0
MOVL C00665 V=800.0 PL=0
MOVL C00666 V=800.0 PL=0
MOVL C00667 V=800.0 PL=0
MOVL C00668 V=800.0 PL=0
MOVL C00669 V=800.0 PL=0
MOVL C00670 V=800.0 PL=0
MOVL C00671 V=800.0 PL=0
MOVL C00672 V=800.0 PL=0
MOVL C00673 V=800.0 PL=0
MOVL C00674 V=800.0 PL=0
MOVL C00675 V=800.0 PL=0
MOVL C00676 V=800.0 PL=0
MOVL C00677 V=800.0 PL=0
MOVL C00678 V=800.0 PL=0
MOVL C00679 V=800.0 PL=0
MOVL C00680 V=800.0 PL=0
MOVL C00681 V=800.0 PL=0
MOVL C00682 V=800.0 PL=0
MOVL C00683 V=800.0 PL=0
MOVL C00684 V=800.0 PL=0
MOVL C00685 V=800.0 PL=0
MOVL C00686 V=800.0 PL=0
MOVL C00687 V=800.0 PL=0
MOVL C00688 V=800.0 PL=0
MOVL C00689 V=800.0 PL=0
MOVL C00690 V=800.0 PL=0
MOVL C00691 V=800.0 PL=0
MOVL C00692 V=800.0 PL=0
MOVL C00693 V=800.0 PL=0
MOVL C00694 V=800.0 PL=0
MOVL C00695 V=800.0 PL=0
MOVL C00696 V=800.0 PL=0
MOVL C00697 V=800.0 PL=0
MOVL C00698 V=800.0 PL=0
MOVL C00699 V=800.0 PL=0
MOVL C00700 V=800.0 PL=0
MOVL C00701 V=800.0 PL=0
MOVL C00702 V=800.0 PL=0
MOVL C00703 V=800.0 PL=0
MOVL C00704 V=800.0 PL=0
MOVL C00705 V=800.0 PL=0
MOVL C00706 V=800.0 PL=0
MOVL C00707 V=800.0 PL=0
MOVL C00708 V=800.0 PL=0
MOVL C00709 V=800.0 PL=0
MOVL C00710 V=800.0 PL=0
MOVL C00711 V=800.0 PL=0
MOVL C00712 V=800.0 PL=0
MOVL C00713 V=800.0 PL=0
MOVL C00714 V=800.0 PL=0
MOVL C00715 V=800.0 PL=0
MOVL C00716 V=800.0 PL=0
MOVL C00717 V=800.0 PL=0
MOVL C00718 V=800.0 PL=0
MOVL C00719 V=800.0 PL=0
MOVL C00720 V=800.0 PL=0
MOVL C00721 V=800.0 PL=0
MOVL C00722 V=800.0 PL=0
MOVL C00723 V=800.0 PL=0
MOVL C00724 V=800.0 PL=0
MOVL C00725 V=800.0 PL=0
MOVL C00726 V=800.0 PL=0
MOVL C00727 V=800.0 PL=0
MOVL C00728 V=800.0 PL=0
MOVL C00729 V=800.0 PL=0
MOVL C00730 V=800.0 PL=0
MOVL C00731 V=800.0 PL=0
MOVL C00732 V=800.0 PL=0
MOVL C00733 V=800.0 PL=0
MOVL C00734 V=800.0 PL=0
MOVL C00735 V=800.0 PL=0
MOVL C00736 V=800.0 PL=0
MOVL C00737 V=800.0 PL=0
MOVL C00738 V=800.0 PL=0
MOVL C00739 V=800.0 PL=0
MOVL C00740 V=800.0 PL=0
MOVL C00741 V=800.0 PL=0
MOVL C00742 V=800.0 PL=0
MOVL C00743 V=800.0 PL=0
MOVL C00744 V=800.0 PL=0
MOVL C00745 V=800.0 PL=0
MOVL C00746 V=800.0 PL=0
MOVL C00747 V=800.0 PL=0
MOVL C00748 V=800.0 PL=0
MOVL C00749 V=800.0 PL=0
MOVL C00750 V=800.0 PL=0
MOVL C00751 V=800.0 PL=0
MOVL C00752 V=800.0 PL=0
MOVL C00753 V=800.0 PL=0
MOVL C00754 V=800.0 PL=0
MOVL C00755 V=800.0 PL=0
MOVL C00756 V=800.0 PL=0
MOVL C00757 V=800.0 PL=0
MOVL C00758 V=800.0 PL=0
MOVL C00759 V=800.0 PL=0
MOVL C00760 V=800.0 PL=0
MOVL C00761 V=800.0 PL=0
MOVL C00762 V=800.0 PL=0
MOVL C00763 V=800.0 PL=0
MOVL C00764 V=800.0 PL=0
MOVL C00765 V=800.0 PL=0
MOVL C00766 V=800.0 PL=0
MOVL C00767 V=800.0 PL=0
MOVL C00768 V=800.0 PL=0
MOVL C00769 V=800.0 PL=0
MOVL C00770 V=800.0 PL=0
MOVL C00771 V=800.0 PL=0
MOVL C00772 V=800.0 PL=0
MOVL C00773 V=800.0 PL=0
MOVL C00774 V=800.0 PL=0
MOVL C00775 V=800.0 PL=0
MOVL C00776 V=800.0 PL=0
MOVL C00777 V=800.0 PL=0
MOVL C00778 V=800.0 PL=0
MOVL C00779 V=800.0 PL=0
MOVL C00780 V=800.0 PL=0
MOVL C00781 V=800.0 PL=0
MOVL C00782 V=800.0 PL=0
MOVL C00783 V=800.0 PL=0
MOVL C00784 V=800.0 PL=0
MOVL C00785 V=800.0 PL=0
MOVL C00786 V=800.0 PL=0
MOVL C00787 V=800.0 PL=0
MOVL C00788 V=800.0 PL=0
MOVL C00789 V=800.0 PL=0
MOVL C00790 V=800.0 PL=0
MOVL C00791 V=800.0 PL=0
MOVL C00792 V=800.0 PL=0
MOVL C00793 V=800.0 PL=0
MOVL C00794 V=800.0 PL=0
MOVL C00795 V=800.0 PL=0
MOVL C00796 V=800.0 PL=0
MOVL C00797 V=800.0 PL=0
MOVL C00798 V=800.0 PL=0
MOVL C00799 V=800.0 PL=0
MOVL C00800 V=800.0 PL=0
MOVL C00801 V=800.0 PL=0
MOVL C00802 V=800.0 PL=0
MOVL C00803 V=800.0 PL=0
MOVL C00804 V=800.0 PL=0
MOVL C00805 V=800.0 PL=0
MOVL C00806 V=800.0 PL=0
MOVL C00807 V=800.0 PL=0
MOVL C00808 V=800.0 PL=0
MOVL C00809 V=800.0 PL=0
MOVL C00810 V=800.0 PL=0
MOVL C00811 V=800.0 PL=0
MOVL C00812 V=800.0 PL=0
MOVL C00813 V=800.0 PL=0
MOVL C00814 V=800.0 PL=0
MOVL C00815 V=800.0 PL=0
MOVL C00816 V=800.0 PL=0
MOVL C00817 V=800.0 PL=0
MOVL C00818 V=800.0 PL=0
MOVL C00819 V=800.0 PL=0
MOVL C00820 V=800.0 PL=0
MOVL C00821 V=800.0 PL=0
MOVL C00822 V=800.0 PL=0
MOVL C00823 V=800.0 PL=0
MOVL C00824 V=800.0 PL=0
MOVL C00825 V=800.0 PL=0
MOVL C00826 V=800.0 PL=0
MOVL C00827 V=800.0 PL=0
MOVL C00828 V=800.0 PL=0
MOVL C00829 V=800.0 PL=0
MOVL C00830 V=800.0 PL=0
MOVL C00831 V=800.0 PL=0
MOVL C00832 V=800.0 PL=0
MOVL C00833 V=800.0 PL=0
MOVL C00834 V=800.0 PL=0
MOVL C00835 V=800.0 PL=0
MOVL C00836 V=800.0 PL=0
MOVL C00837 V=800.0 PL=0
MOVL C00838 V=800.0 PL=0
MOVL C00839 V=800.0 PL=0
MOVL C00840 V=800.0 PL=0
MOVL C00841 V=800.0 PL=0
MOVL C00842 V=800.0 PL=0
MOVL C00843 V=800.0 PL=0
MOVL C00844 V=800.0 PL=0
MOVL C00845 V=800.0 PL=0
MOVL C00846 V=800.0 PL=0
MOVL C00847 V=800.0 PL=0
MOVL C00848 V=800.0 PL=0
MOVL C00849 V=800.0 PL=0
MOVL C00850 V=800.0 PL=0
MOVL C00851 V=800.0 PL=0
MOVL C00852 V=800.0 PL=0
MOVL C00853 V=800.0 PL=0
MOVL C00854 V=800.0 PL=0
MOVL C00855 V=800.0 PL=0
MOVL C00856 V=800.0 PL=0
MOVL C00857 V=800.0 PL=0
MOVL C00858 V=800.0 PL=0
MOVL C00859 V=800.0 PL=0
MOVL C00860 V=800.0 PL=0
MOVL C00861 V=800.0 PL=0
MOVL C00862 V=800.0 PL=0
MOVL C00863 V=800.0 PL=0
MOVL C00864 V=800.0 PL=0
MOVL C00865 V=800.0 PL=0
MOVL C00866 V=800.0 PL=0
MOVL C00867 V=800.0 PL=0
MOVL C00868 V=800.0 PL=0
MOVL C00869 V=800.0 PL=0
MOVL C00870 V=800.0 PL=0
MOVL C00871 V=800.0 PL=0
MOVL C00872 V=800.0 PL=0
MOVL C00873 V=800.0 PL=0
MOVL C00874 V=800.0 PL=0
MOVL C00875 V=800.0 PL=0
MOVL C00876 V=800.0 PL=0
MOVL C00877 V=800.0 PL=0
MOVL C00878 V=800.0 PL=0
MOVL C00879 V=800.0 PL=0
MOVL C00880 V=800.0 PL=0
MOVL C00881 V=800.0 PL=0
MOVL C00882 V=800.0 PL=0
MOVL C00883 V=800.0 PL=0
MOVL C00884 V=800.0 PL=0
MOVL C00885 V=800.0 PL=0
MOVL C00886 V=800.0 PL=0
MOVL C00887 V=800.0 PL=0
MOVL C00888 V=800.0 PL=0
MOVL C00889 V=800.0 PL=0
MOVL C00890 V=800.0 PL=0
MOVL C00891 V=800.0 PL=0
MOVL C00892 V=800.0 PL=0
MOVL C00893 V=800.0 PL=0
MOVL C00894 V=800.0 PL=0
MOVL C00895 V=800.0 PL=0
MOVL C00896 V=800.0 PL=0
MOVL C00897 V=800.0 PL=0
MOVL C00898 V=800.0 PL=0
MOVL C00899 V=800.0 PL=0
MOVL C00900 V=800.0 PL=0
MOVL C00901 V=800.0 PL=0
MOVL C00902 V=800.0 PL=0
MOVL C00903 V=800.0 PL=0
MOVL C00904 V=800.0 PL=0
MOVL C00905 V=800.0 PL=0
MOVL C00906 V=800.0 PL=0
MOVL C00907 V=800.0 PL=0
MOVL C00908 V=800.0 PL=0
MOVL C00909 V=800.0 PL=0
MOVL C00910 V=800.0 PL=0
MOVL C00911 V=800.0 PL=0
MOVL C00912 V=800.0 PL=0
MOVL C00913 V=800.0 PL=0
MOVL C00914 V=800.0 PL=0
MOVL C00915 V=800.0 PL=0
MOVL C00916 V=800.0 PL=0
MOVL C00917 V=800.0 PL=0
MOVL C00918 V=800.0 PL=0
MOVL C00919 V=800.0 PL=0
MOVL C00920 V=800.0 PL=0
MOVL C00921 V=800.0 PL=0
MOVL C00922 V=800.0 PL=0
MOVL C00923 V=800.0 PL=0
MOVL C00924 V=800.0 PL=0
MOVL C00925 V=800.0 PL=0
MOVL C00926 V=800.0 PL=0
MOVL C00927 V=800.0 PL=0
MOVL C00928 V=800.0 PL=0
MOVL C00929 V=800.0 PL=0
MOVL C00930 V=800.0 PL=0
MOVL C00931 V=800.0 PL=0
MOVL C00932 V=800.0 PL=0
MOVL C00933 V=800.0 PL=0
MOVL C00934 V=800.0 PL=0
MOVL C00935 V=800.0 PL=0
MOVL C00936 V=800.0 PL=0
MOVL C00937 V=800.0 PL=0
MOVL C00938 V=800.0 PL=0
MOVL C00939 V=800.0 PL=0
MOVL C00940 V=800.0 PL=0
MOVL C00941 V=800.0 PL=0
MOVL C00942 V=800.0 PL=0
MOVL C00943 V=800.0 PL=0
MOVL C00944 V=800.0 PL=0
MOVL C00945 V=800.0 PL=0
MOVL C00946 V=800.0 PL=0
MOVL C00947 V=800.0 PL=0
MOVL C00948 V=800.0 PL=0
MOVL C00949 V=800.0 PL=0
MOVL C00950 V=800.0 PL=0
MOVL C00951 V=800.0 PL=0
MOVL C00952 V=800.0 PL=0
MOVL C00953 V=800.0 PL=0
MOVL C00954 V=800.0 PL=0
MOVL C00955 V=800.0 PL=0
MOVL C00956 V=800.0 PL=0
MOVL C00957 V=800.0 PL=0
MOVL C00958 V=800.0 PL=0
MOVL C00959 V=800.0 PL=0
MOVL C00960 V=800.0 PL=0
MOVL C00961 V=800.0 PL=0
MOVL C00962 V=800.0 PL=0
MOVL C00963 V=800.0 PL=0
MOVL C00964 V=800.0 PL=0
MOVL C00965 V=800.0 PL=0
MOVL C00966 V=800.0 PL=0
MOVL C00967 V=800.0 PL=0
MOVL C00968 V=800.0 PL=0
MOVL C00969 V=800.0 PL=0
MOVL C00970 V=800.0 PL=0
MOVL C00971 V=800.0 PL=0
MOVL C00972 V=800.0 PL=0
MOVL C00973 V=800.0 PL=0
MOVL C00974 V=800.0 PL=0
MOVL C00975 V=800.0 PL=0
MOVL C00976 V=800.0 PL=0
MOVL C00977 V=800.0 PL=0
MOVL C00978 V=800.0 PL=0
MOVL C00979 V=800.0 PL=0
MOVL C00980 V=800.0 PL=0
MOVL C00981 V=800.0 PL=0
MOVL C00982 V=800.0 PL=0
MOVL C00983 V=800.0 PL=0
MOVL C00984 V=800.0 PL=0
MOVL C00985 V=800.0 PL=0
MOVL C00986 V=800.0 PL=0
MOVL C00987 V=800.0 PL=0
MOVL C00988 V=800.0 PL=0
MOVL C00989 V=800.0 PL=0
MOVL C00990 V=800.0 PL=0
MOVL C00991 V=800.0 PL=0
MOVL C00992 V=800.0 PL=0
MOVL C00993 V=800.0 PL=0
MOVL C00994 V=800.0 PL=0
MOVL C00995 V=800.0 PL=0
MOVL C00996 V=800.0 PL=0
MOVL C00997 V=800.0 PL=0
MOVL C00998 V=800.0 PL=0
MOVL C00999 V=800.0 PL=0
MOVL C01000 V=800.0 PL=0
MOVL C01001 V=800.0 PL=0
MOVL C01002 V=800.0 PL=0
MOVL C01003 V=800.0 PL=0
MOVL C01004 V=800.0 PL=0
MOVL C01005 V=800.0 PL=0
MOVL C01006 V=800.0 PL=0
MOVL C01007 V=800.0 PL=0
MOVL C01008 V=800.0 PL=0
MOVL C01009 V=800.0 PL=0
MOVL C01010 V=800.0 PL=0
MOVL C01011 V=800.0 PL=0
MOVL C01012 V=800.0 PL=0
MOVL C01013 V=800.0 PL=0
MOVL C01014 V=800.0 PL=0
MOVL C01015 V=800.0 PL=0
MOVL C01016 V=800.0 PL=0
MOVL C01017 V=800.0 PL=0
MOVL C01018 V=800.0 PL=0
MOVL C01019 V=800.0 PL=0
MOVL C01020 V=800.0 PL=0
MOVL C01021 V=800.0 PL=0
MOVL C01022 V=800.0 PL=0
MOVL C01023 V=800.0 PL=0
MOVL C01024 V=800.0 PL=0
MOVL C01025 V=800.0 PL=0
MOVL C01026 V=800.0 PL=0
MOVL C01027 V=800.0 PL=0
MOVL C01028 V=800.0 PL=0
MOVL C01029 V=800.0 PL=0
MOVL C01030 V=800.0 PL=0
MOVL C01031 V=800.0 PL=0
MOVL C01032 V=800.0 PL=0
MOVL C01033 V=800.0 PL=0
MOVL C01034 V=800.0 PL=0
MOVL C01035 V=800.0 PL=0
MOVL C01036 V=800.0 PL=0
MOVL C01037 V=800.0 PL=0
MOVL C01038 V=800.0 PL=0
MOVL C01039 V=800.0 PL=0
MOVL C01040 V=800.0 PL=0
MOVL C01041 V=800.0 PL=0
MOVL C01042 V=800.0 PL=0
MOVL C01043 V=800.0 PL=0
MOVL C01044 V=800.0 PL=0
MOVL C01045 V=800.0 PL=0
MOVL C01046 V=800.0 PL=0
MOVL C01047 V=800.0 PL=0
MOVL C01048 V=800.0 PL=0
MOVL C01049 V=800.0 PL=0
MOVL C01050 V=800.0 PL=0
MOVL C01051 V=800.0 PL=0
MOVL C01052 V=800.0 PL=0
MOVL C01053 V=800.0 PL=0
MOVL C01054 V=800.0 PL=0
MOVL C01055 V=800.0 PL=0
MOVL C01056 V=800.0 PL=0
MOVL C01057 V=800.0 PL=0
MOVL C01058 V=800.0 PL=0
MOVL C01059 V=800.0 PL=0
MOVL C01060 V=800.0 PL=0
MOVL C01061 V=800.0 PL=0
MOVL C01062 V=800.0 PL=0
MOVL C01063 V=800.0 PL=0
MOVL C01064 V=800.0 PL=0
MOVL C01065 V=800.0 PL=0
MOVL C01066 V=800.0 PL=0
MOVL C01067 V=800.0 PL=0
MOVL C01068 V=800.0 PL=0
MOVL C01069 V=800.0 PL=0
MOVL C01070 V=800.0 PL=0
MOVL C01071 V=800.0 PL=0
MOVL C01072 V=800.0 PL=0
MOVL C01073 V=800.0 PL=0
MOVL C01074 V=800.0 PL=0
MOVL C01075 V=800.0 PL=0
MOVL C01076 V=800.0 PL=0
MOVL C01077 V=800.0 PL=0
MOVL C01078 V=800.0 PL=0
MOVL C01079 V=800.0 PL=0
MOVL C01080 V=800.0 PL=0
MOVL C01081 V=800.0 PL=0
MOVL C01082 V=800.0 PL=0
MOVL C01083 V=800.0 PL=0
MOVL C01084 V=800.0 PL=0
MOVL C01085 V=800.0 PL=0
MOVL C01086 V=800.0 PL=0
MOVL C01087 V=800.0 PL=0
MOVL C01088 V=800.0 PL=0
MOVL C01089 V=800.0 PL=0
MOVL C01090 V=800.0 PL=0
MOVL C01091 V=800.0 PL=0
MOVL C01092 V=800.0 PL=0
MOVL C01093 V=800.0 PL=0
MOVL C01094 V=800.0 PL=0
MOVL C01095 V=800.0 PL=0
MOVL C01096 V=800.0 PL=0
MOVL C01097 V=800.0 PL=0
MOVL C01098 V=800.0 PL=0
MOVL C01099 V=800.0 PL=0
MOVL C01100 V=800.0 PL=0
MOVL C01101 V=800.0 PL=0
MOVL C01102 V=800.0 PL=0
MOVL C01103 V=800.0 PL=0
MOVL C01104 V=800.0 PL=0
MOVL C01105 V=800.0 PL=0
MOVL C01106 V=800.0 PL=0
MOVL C01107 V=800.0 PL=0
MOVL C01108 V=800.0 PL=0
MOVL C01109 V=800.0 PL=0
MOVL C01110 V=800.0 PL=0
MOVL C01111 V=800.0 PL=0
MOVL C01112 V=800.0 PL=0
MOVL C01113 V=800.0 PL=0
MOVL C01114 V=800.0 PL=0
MOVL C01115 V=800.0 PL=0
MOVL C01116 V=800.0 PL=0
MOVL C01117 V=800.0 PL=0
MOVL C01118 V=800.0 PL=0
MOVL C01119 V=800.0 PL=0
MOVL C01120 V=800.0 PL=0
MOVL C01121 V=800.0 PL=0
MOVL C01122 V=800.0 PL=0
MOVL C01123 V=800.0 PL=0
MOVL C01124 V=800.0 PL=0
MOVL C01125 V=800.0 PL=0
MOVL C01126 V=800.0 PL=0
MOVL C01127 V=800.0 PL=0
MOVL C01128 V=800.0 PL=0
MOVL C01129 V=800.0 PL=0
MOVL C01130 V=800.0 PL=0
MOVL C01131 V=800.0 PL=0
MOVL C01132 V=800.0 PL=0
MOVL C01133 V=800.0 PL=0
MOVL C01134 V=800.0 PL=0
MOVL C01135 V=800.0 PL=0
MOVL C01136 V=800.0 PL=0
MOVL C01137 V=800.0 PL=0
MOVL C01138 V=800.0 PL=0
MOVL C01139 V=800.0 PL=0
MOVL C01140 V=800.0 PL=0
MOVL C01141 V=800.0 PL=0
MOVL C01142 V=800.0 PL=0
MOVL C01143 V=800.0 PL=0
MOVL C01144 V=800.0 PL=0
MOVL C01145 V=800.0 PL=0
MOVL C01146 V=800.0 PL=0
MOVL C01147 V=800.0 PL=0
MOVL C01148 V=800.0 PL=0
MOVL C01149 V=800.0 PL=0
MOVL C01150 V=800.0 PL=0
MOVL C01151 V=800.0 PL=0
MOVL C01152 V=800.0 PL=0
MOVL C01153 V=800.0 PL=0
MOVL C01154 V=800.0 PL=0
MOVL C01155 V=800.0 PL=0
MOVL C01156 V=800.0 PL=0
MOVL C01157 V=800.0 PL=0
MOVL C01158 V=800.0 PL=0
MOVL C01159 V=800.0 PL=0
MOVL C01160 V=800.0 PL=0
MOVL C01161 V=800.0 PL=0
MOVL C01162 V=800.0 PL=0
MOVL C01163 V=800.0 PL=0
MOVL C01164 V=800.0 PL=0
MOVL C01165 V=800.0 PL=0
MOVL C01166 V=800.0 PL=0
MOVL C01167 V=800.0 PL=0
MOVL C01168 V=800.0 PL=0
MOVL C01169 V=800.0 PL=0
MOVL C01170 V=800.0 PL=0
MOVL C01171 V=800.0 PL=0
MOVL C01172 V=800.0 PL=0
MOVL C01173 V=800.0 PL=0
MOVL C01174 V=800.0 PL=0
MOVL C01175 V=800.0 PL=0
MOVL C01176 V=800.0 PL=0
MOVL C01177 V=800.0 PL=0
MOVL C01178 V=800.0 PL=0
MOVL C01179 V=800.0 PL=0
MOVL C01180 V=800.0 PL=0
MOVL C01181 V=800.0 PL=0
MOVL C01182 V=800.0 PL=0
MOVL C01183 V=800.0 PL=0
MOVL C01184 V=800.0 PL=0
MOVL C01185 V=800.0 PL=0
MOVL C01186 V=800.0 PL=0
MOVL C01187 V=800.0 PL=0
MOVL C01188 V=800.0 PL=0
MOVL C01189 V=800.0 PL=0
MOVL C01190 V=800.0 PL=0
MOVL C01191 V=800.0 PL=0
MOVL C01192 V=800.0 PL=0
MOVL C01193 V=800.0 PL=0
MOVL C01194 V=800.0 PL=0
MOVL C01195 V=800.0 PL=0
MOVL C01196 V=800.0 PL=0
MOVL C01197 V=800.0 PL=0
MOVL C01198 V=800.0 PL=0
MOVL C01199 V=800.0 PL=0
MOVL C01200 V=800.0 PL=0
MOVL C01201 V=800.0 PL=0
MOVL C01202 V=800.0 PL=0
MOVL C01203 V=800.0 PL=0
MOVL C01204 V=800.0 PL=0
MOVL C01205 V=800.0 PL=0
MOVL C01206 V=800.0 PL=0
MOVL C01207 V=800.0 PL=0
MOVL C01208 V=800.0 PL=0
MOVL C01209 V=800.0 PL=0
MOVL C01210 V=800.0 PL=0
MOVL C01211 V=800.0 PL=0
MOVL C01212 V=800.0 PL=0
MOVL C01213 V=800.0 PL=0
MOVL C01214 V=800.0 PL=0
MOVL C01215 V=800.0 PL=0
MOVL C01216 V=800.0 PL=0
MOVL C01217 V=800.0 PL=0
MOVL C01218 V=800.0 PL=0
MOVL C01219 V=800.0 PL=0
MOVL C01220 V=800.0 PL=0
MOVL C01221 V=800.0 PL=0
MOVL C01222 V=800.0 PL=0
MOVL C01223 V=800.0 PL=0
MOVL C01224 V=800.0 PL=0
MOVL C01225 V=800.0 PL=0
MOVL C01226 V=800.0 PL=0
MOVL C01227 V=800.0 PL=0
MOVL C01228 V=800.0 PL=0
MOVL C01229 V=800.0 PL=0
MOVL C01230 V=800.0 PL=0
MOVL C01231 V=800.0 PL=0
MOVL C01232 V=800.0 PL=0
MOVL C01233 V=800.0 PL=0
MOVL C01234 V=800.0 PL=0
MOVL C01235 V=800.0 PL=0
MOVL C01236 V=800.0 PL=0
MOVL C01237 V=800.0 PL=0
MOVL C01238 V=800.0 PL=0
MOVL C01239 V=800.0 PL=0
MOVL C01240 V=800.0 PL=0
MOVL C01241 V=800.0 PL=0
MOVL C01242 V=800.0 PL=0
MOVL C01243 V=800.0 PL=0
MOVL C01244 V=800.0 PL=0
MOVL C01245 V=800.0 PL=0
MOVL C01246 V=800.0 PL=0
MOVL C01247 V=800.0 PL=0
MOVL C01248 V=800.0 PL=0
MOVL C01249 V=800.0 PL=0
MOVL C01250 V=800.0 PL=0
MOVL C01251 V=800.0 PL=0
MOVL C01252 V=800.0 PL=0
MOVL C01253 V=800.0 PL=0
MOVL C01254 V=800.0 PL=0
MOVL C01255 V=800.0 PL=0
MOVL C01256 V=800.0 PL=0
MOVL C01257 V=800.0 PL=0
MOVL C01258 V=800.0 PL=0
MOVL C01259 V=800.0 PL=0
MOVL C01260 V=800.0 PL=0
MOVL C01261 V=800.0 PL=0
MOVL C01262 V=800.0 PL=0
MOVL C01263 V=800.0 PL=0
MOVL C01264 V=800.0 PL=0
MOVL C01265 V=800.0 PL=0
MOVL C01266 V=800.0 PL=0
MOVL C01267 V=800.0 PL=0
MOVL C01268 V=800.0 PL=0
MOVL C01269 V=800.0 PL=0
MOVL C01270 V=800.0 PL=0
MOVL C01271 V=800.0 PL=0
MOVL C01272 V=800.0 PL=0
MOVL C01273 V=800.0 PL=0
MOVL C01274 V=800.0 PL=0
MOVL C01275 V=800.0 PL=0
MOVL C01276 V=800.0 PL=0
MOVL C01277 V=800.0 PL=0
MOVL C01278 V=800.0 PL=0
MOVL C01279 V=800.0 PL=0
MOVL C01280 V=800.0 PL=0
MOVL C01281 V=800.0 PL=0
MOVL C01282 V=800.0 PL=0
MOVL C01283 V=800.0 PL=0
MOVL C01284 V=800.0 PL=0
MOVL C01285 V=800.0 PL=0
MOVL C01286 V=800.0 PL=0
MOVL C01287 V=800.0 PL=0
MOVL C01288 V=800.0 PL=0
MOVL C01289 V=800.0 PL=0
MOVL C01290 V=800.0 PL=0
MOVL C01291 V=800.0 PL=0
MOVL C01292 V=800.0 PL=0
MOVL C01293 V=800.0 PL=0
MOVL C01294 V=800.0 PL=0
MOVL C01295 V=800.0 PL=0
MOVL C01296 V=800.0 PL=0
MOVL C01297 V=800.0 PL=0
MOVL C01298 V=800.0 PL=0
MOVL C01299 V=800.0 PL=0
MOVL C01300 V=800.0 PL=0
MOVL C01301 V=800.0 PL=0
MOVL C01302 V=800.0 PL=0
MOVL C01303 V=800.0 PL=0
MOVL C01304 V=800.0 PL=0
MOVL C01305 V=800.0 PL=0
MOVL C01306 V=800.0 PL=0
MOVL C01307 V=800.0 PL=0
MOVL C01308 V=800.0 PL=0
MOVL C01309 V=800.0 PL=0
MOVL C01310 V=800.0 PL=0
MOVL C01311 V=800.0 PL=0
MOVL C01312 V=800.0 PL=0
MOVL C01313 V=800.0 PL=0
MOVL C01314 V=800.0 PL=0
MOVL C01315 V=800.0 PL=0
MOVL C01316 V=800.0 PL=0
MOVL C01317 V=800.0 PL=0
MOVL C01318 V=800.0 PL=0
MOVL C01319 V=800.0 PL=0
MOVL C01320 V=800.0 PL=0
MOVL C01321 V=800.0 PL=0
MOVL C01322 V=800.0 PL=0
MOVL C01323 V=800.0 PL=0
MOVL C01324 V=800.0 PL=0
MOVL C01325 V=800.0 PL=0
MOVL C01326 V=800.0 PL=0
MOVL C01327 V=800.0 PL=0
MOVL C01328 V=800.0 PL=0
MOVL C01329 V=800.0 PL=0
MOVL C01330 V=800.0 PL=0
MOVL C01331 V=800.0 PL=0
MOVL C01332 V=800.0 PL=0
MOVL C01333 V=800.0 PL=0
MOVL C01334 V=800.0 PL=0
MOVL C01335 V=800.0 PL=0
MOVL C01336 V=800.0 PL=0
MOVL C01337 V=800.0 PL=0
MOVL C01338 V=800.0 PL=0
MOVL C01339 V=800.0 PL=0
MOVL C01340 V=800.0 PL=0
MOVL C01341 V=800.0 PL=0
MOVL C01342 V=800.0 PL=0
MOVL C01343 V=800.0 PL=0
MOVL C01344 V=800.0 PL=0
MOVL C01345 V=800.0 PL=0
MOVL C01346 V=800.0 PL=0
MOVL C01347 V=800.0 PL=0
MOVL C01348 V=800.0 PL=0
MOVL C01349 V=800.0 PL=0
MOVL C01350 V=800.0 PL=0
MOVL C01351 V=800.0 PL=0
MOVL C01352 V=800.0 PL=0
MOVL C01353 V=800.0 PL=0
MOVL C01354 V=800.0 PL=0
MOVL C01355 V=800.0 PL=0
MOVL C01356 V=800.0 PL=0
MOVL C01357 V=800.0 PL=0
MOVL C01358 V=800.0 PL=0
MOVL C01359 V=800.0 PL=0
MOVL C01360 V=800.0 PL=0
MOVL C01361 V=800.0 PL=0
MOVL C01362 V=800.0 PL=0
MOVL C01363 V=800.0 PL=0
MOVL C01364 V=800.0 PL=0
MOVL C01365 V=800.0 PL=0
MOVL C01366 V=800.0 PL=0
MOVL C01367 V=800.0 PL=0
MOVL C01368 V=800.0 PL=0
MOVL C01369 V=800.0 PL=0
MOVL C01370 V=800.0 PL=0
MOVL C01371 V=800.0 PL=0
MOVL C01372 V=800.0 PL=0
MOVL C01373 V=800.0 PL=0
MOVL C01374 V=800.0 PL=0
MOVL C01375 V=800.0 PL=0
MOVL C01376 V=800.0 PL=0
MOVL C01377 V=800.0 PL=0
MOVL C01378 V=800.0 PL=0
MOVL C01379 V=800.0 PL=0
MOVL C01380 V=800.0 PL=0
MOVL C01381 V=800.0 PL=0
MOVL C01382 V=800.0 PL=0
MOVL C01383 V=800.0 PL=0
MOVL C01384 V=800.0 PL=0
MOVL C01385 V=800.0 PL=0
MOVL C01386 V=800.0 PL=0
MOVL C01387 V=800.0 PL=0
MOVL C01388 V=800.0 PL=0
MOVL C01389 V=800.0 PL=0
MOVL C01390 V=800.0 PL=0
MOVL C01391 V=800.0 PL=0
MOVL C01392 V=800.0 PL=0
MOVL C01393 V=800.0 PL=0
MOVL C01394 V=800.0 PL=0
MOVL C01395 V=800.0 PL=0
MOVL C01396 V=800.0 PL=0
MOVL C01397 V=800.0 PL=0
MOVL C01398 V=800.0 PL=0
MOVL C01399 V=800.0 PL=0
MOVL C01400 V=800.0 PL=0
MOVL C01401 V=800.0 PL=0
MOVL C01402 V=800.0 PL=0
MOVL C01403 V=800.0 PL=0
MOVL C01404 V=800.0 PL=0
MOVL C01405 V=800.0 PL=0
MOVL C01406 V=800.0 PL=0
MOVL C01407 V=800.0 PL=0
MOVL C01408 V=800.0 PL=0
MOVL C01409 V=800.0 PL=0
MOVL C01410 V=800.0 PL=0
MOVL C01411 V=800.0 PL=0
MOVL C01412 V=800.0 PL=0
MOVL C01413 V=800.0 PL=0
MOVL C01414 V=800.0 PL=0
MOVL C01415 V=800.0 PL=0
MOVL C01416 V=800.0 PL=0
MOVL C01417 V=800.0 PL=0
MOVL C01418 V=800.0 PL=0
MOVL C01419 V=800.0 PL=0
MOVL C01420 V=800.0 PL=0
MOVL C01421 V=800.0 PL=0
MOVL C01422 V=800.0 PL=0
MOVL C01423 V=800.0 PL=0
MOVL C01424 V=800.0 PL=0
MOVL C01425 V=800.0 PL=0
MOVL C01426 V=800.0 PL=0
MOVL C01427 V=800.0 PL=0
MOVL C01428 V=800.0 PL=0
MOVL C01429 V=800.0 PL=0
MOVL C01430 V=800.0 PL=0
MOVL C01431 V=800.0 PL=0
MOVL C01432 V=800.0 PL=0
MOVL C01433 V=800.0 PL=0
MOVL C01434 V=800.0 PL=0
MOVL C01435 V=800.0 PL=0
MOVL C01436 V=800.0 PL=0
MOVL C01437 V=800.0 PL=0
MOVL C01438 V=800.0 PL=0
MOVL C01439 V=800.0 PL=0
MOVL C01440 V=800.0 PL=0
MOVL C01441 V=800.0 PL=0
MOVL C01442 V=800.0 PL=0
MOVL C01443 V=800.0 PL=0
MOVL C01444 V=800.0 PL=0
MOVL C01445 V=800.0 PL=0
MOVL C01446 V=800.0 PL=0
MOVL C01447 V=800.0 PL=0
MOVL C01448 V=800.0 PL=0
MOVL C01449 V=800.0 PL=0
MOVL C01450 V=800.0 PL=0
MOVL C01451 V=800.0 PL=0
MOVL C01452 V=800.0 PL=0
MOVL C01453 V=800.0 PL=0
MOVL C01454 V=800.0 PL=0
MOVL C01455 V=800.0 PL=0
MOVL C01456 V=800.0 PL=0
MOVL C01457 V=800.0 PL=0
MOVL C01458 V=800.0 PL=0
MOVL C01459 V=800.0 PL=0
MOVL C01460 V=800.0 PL=0
MOVL C01461 V=800.0 PL=0
MOVL C01462 V=800.0 PL=0
MOVL C01463 V=800.0 PL=0
MOVL C01464 V=800.0 PL=0
MOVL C01465 V=800.0 PL=0
MOVL C01466 V=800.0 PL=0
MOVL C01467 V=800.0 PL=0
MOVL C01468 V=800.0 PL=0
MOVL C01469 V=800.0 PL=0
MOVL C01470 V=800.0 PL=0
MOVL C01471 V=800.0 PL=0
MOVL C01472 V=800.0 PL=0
MOVL C01473 V=800.0 PL=0
MOVL C01474 V=800.0 PL=0
MOVL C01475 V=800.0 PL=0
MOVL C01476 V=800.0 PL=0
MOVL C01477 V=800.0 PL=0
MOVL C01478 V=800.0 PL=0
MOVL C01479 V=800.0 PL=0
MOVL C01480 V=800.0 PL=0
MOVL C01481 V=800.0 PL=0
MOVL C01482 V=800.0 PL=0
MOVL C01483 V=800.0 PL=0
MOVL C01484 V=800.0 PL=0
MOVL C01485 V=800.0 PL=0
MOVL C01486 V=800.0 PL=0
MOVL C01487 V=800.0 PL=0
MOVL C01488 V=800.0 PL=0
MOVL C01489 V=800.0 PL=0
MOVL C01490 V=800.0 PL=0
MOVL C01491 V=800.0 PL=0
MOVL C01492 V=800.0 PL=0
MOVL C01493 V=800.0 PL=0
MOVL C01494 V=800.0 PL=0
MOVL C01495 V=800.0 PL=0
MOVL C01496 V=800.0 PL=0
MOVL C01497 V=800.0 PL=0
MOVL C01498 V=800.0 PL=0
MOVL C01499 V=800.0 PL=0
MOVL C01500 V=800.0 PL=0
MOVL C01501 V=800.0 PL=0
MOVL C01502 V=800.0 PL=0
MOVL C01503 V=800.0 PL=0
MOVL C01504 V=800.0 PL=0
MOVL C01505 V=800.0 PL=0
MOVL C01506 V=800.0 PL=0
MOVL C01507 V=800.0 PL=0
MOVL C01508 V=800.0 PL=0
MOVL C01509 V=800.0 PL=0
MOVL C01510 V=800.0 PL=0
MOVL C01511 V=800.0 PL=0
MOVL C01512 V=800.0 PL=0
MOVL C01513 V=800.0 PL=0
MOVL C01514 V=800.0 PL=0
MOVL C01515 V=800.0 PL=0
MOVL C01516 V=800.0 PL=0
MOVL C01517 V=800.0 PL=0
MOVL C01518 V=800.0 PL=0
MOVL C01519 V=800.0 PL=0
MOVL C01520 V=800.0 PL=0
MOVL C01521 V=800.0 PL=0
MOVL C01522 V=800.0 PL=0
MOVL C01523 V=800.0 PL=0
MOVL C01524 V=800.0 PL=0
MOVL C01525 V=800.0 PL=0
MOVL C01526 V=800.0 PL=0
MOVL C01527 V=800.0 PL=0
MOVL C01528 V=800.0 PL=0
MOVL C01529 V=800.0 PL=0
MOVL C01530 V=800.0 PL=0
MOVL C01531 V=800.0 PL=0
MOVL C01532 V=800.0 PL=0
MOVL C01533 V=800.0 PL=0
MOVL C01534 V=800.0 PL=0
MOVL C01535 V=800.0 PL=0
MOVL C01536 V=800.0 PL=0
MOVL C01537 V=800.0 PL=0
MOVL C01538 V=800.0 PL=0
MOVL C01539 V=800.0 PL=0
MOVL C01540 V=800.0 PL=0
MOVL C01541 V=800.0 PL=0
MOVL C01542 V=800.0 PL=0
MOVL C01543 V=800.0 PL=0
MOVL C01544 V=800.0 PL=0
MOVL C01545 V=800.0 PL=0
MOVL C01546 V=800.0 PL=0
MOVL C01547 V=800.0 PL=0
MOVL C01548 V=800.0 PL=0
MOVL C01549 V=800.0 PL=0
MOVL C01550 V=800.0 PL=0
MOVL C01551 V=800.0 PL=0
MOVL C01552 V=800.0 PL=0
MOVL C01553 V=800.0 PL=0
MOVL C01554 V=800.0 PL=0
MOVL C01555 V=800.0 PL=0
MOVL C01556 V=800.0 PL=0
MOVL C01557 V=800.0 PL=0
MOVL C01558 V=800.0 PL=0
MOVL C01559 V=800.0 PL=0
MOVL C01560 V=800.0 PL=0
MOVL C01561 V=800.0 PL=0
MOVL C01562 V=800.0 PL=0
MOVL C01563 V=800.0 PL=0
MOVL C01564 V=800.0 PL=0
MOVL C01565 V=800.0 PL=0
MOVL C01566 V=800.0 PL=0
MOVL C01567 V=800.0 PL=0
MOVL C01568 V=800.0 PL=0
MOVL C01569 V=800.0 PL=0
MOVL C01570 V=800.0 PL=0
MOVL C01571 V=800.0 PL=0
MOVL C01572 V=800.0 PL=0
MOVL C01573 V=800.0 PL=0
MOVL C01574 V=800.0 PL=0
MOVL C01575 V=800.0 PL=0
MOVL C01576 V=800.0 PL=0
MOVL C01577 V=800.0 PL=0
MOVL C01578 V=800.0 PL=0
MOVL C01579 V=800.0 PL=0
MOVL C01580 V=800.0 PL=0
MOVL C01581 V=800.0 PL=0
MOVL C01582 V=800.0 PL=0
MOVL C01583 V=800.0 PL=0
MOVL C01584 V=800.0 PL=0
MOVL C01585 V=800.0 PL=0
MOVL C01586 V=800.0 PL=0
MOVL C01587 V=800.0 PL=0
MOVL C01588 V=800.0 PL=0
MOVL C01589 V=800.0 PL=0
MOVL C01590 V=800.0 PL=0
MOVL C01591 V=800.0 PL=0
MOVL C01592 V=800.0 PL=0
MOVL C01593 V=800.0 PL=0
MOVL C01594 V=800.0 PL=0
MOVL C01595 V=800.0 PL=0
MOVL C01596 V=800.0 PL=0
MOVL C01597 V=800.0 PL=0
MOVL C01598 V=800.0 PL=0
MOVL C01599 V=800.0 PL=0
MOVL C01600 V=800.0 PL=0
MOVL C01601 V=800.0 PL=0
MOVL C01602 V=800.0 PL=0
MOVL C01603 V=800.0 PL=0
MOVL C01604 V=800.0 PL=0
MOVL C01605 V=800.0 PL=0
MOVL C01606 V=800.0 PL=0
MOVL C01607 V=800.0 PL=0
MOVL C01608 V=800.0 PL=0
MOVL C01609 V=800.0 PL=0
MOVL C01610 V=800.0 PL=0
MOVL C01611 V=800.0 PL=0
MOVL C01612 V=800.0 PL=0
MOVL C01613 V=800.0 PL=0
MOVL C01614 V=800.0 PL=0
MOVL C01615 V=800.0 PL=0
MOVL C01616 V=800.0 PL=0
MOVL C01617 V=800.0 PL=0
MOVL C01618 V=800.0 PL=0
MOVL C01619 V=800.0 PL=0
MOVL C01620 V=800.0 PL=0
MOVL C01621 V=800.0 PL=0
MOVL C01622 V=800.0 PL=0
MOVL C01623 V=800.0 PL=0
MOVL C01624 V=800.0 PL=0
MOVL C01625 V=800.0 PL=0
MOVL C01626 V=800.0 PL=0
MOVL C01627 V=800.0 PL=0
MOVL C01628 V=800.0 PL=0
MOVL C01629 V=800.0 PL=0
MOVL C01630 V=800.0 PL=0
MOVL C01631 V=800.0 PL=0
MOVL C01632 V=800.0 PL=0
MOVL C01633 V=800.0 PL=0
MOVL C01634 V=800.0 PL=0
MOVL C01635 V=800.0 PL=0
MOVL C01636 V=800.0 PL=0
MOVL C01637 V=800.0 PL=0
MOVL C01638 V=800.0 PL=0
MOVL C01639 V=800.0 PL=0
MOVL C01640 V=800.0 PL=0
MOVL C01641 V=800.0 PL=0
MOVL C01642 V=800.0 PL=0
MOVL C01643 V=800.0 PL=0
MOVL C01644 V=800.0 PL=0
MOVL C01645 V=800.0 PL=0
MOVL C01646 V=800.0 PL=0
MOVL C01647 V=800.0 PL=0
MOVL C01648 V=800.0 PL=0
MOVL C01649 V=800.0 PL=0
MOVL C01650 V=800.0 PL=0
MOVL C01651 V=800.0 PL=0
MOVL C01652 V=800.0 PL=0
MOVL C01653 V=800.0 PL=0
MOVL C01654 V=800.0 PL=0
MOVL C01655 V=800.0 PL=0
MOVL C01656 V=800.0 PL=0
MOVL C01657 V=800.0 PL=0
MOVL C01658 V=800.0 PL=0
MOVL C01659 V=800.0 PL=0
MOVL C01660 V=800.0 PL=0
MOVL C01661 V=800.0 PL=0
MOVL C01662 V=800.0 PL=0
MOVL C01663 V=800.0 PL=0
MOVL C01664 V=800.0 PL=0
MOVL C01665 V=800.0 PL=0
MOVL C01666 V=800.0 PL=0
MOVL C01667 V=800.0 PL=0
MOVL C01668 V=800.0 PL=0
MOVL C01669 V=800.0 PL=0
MOVL C01670 V=800.0 PL=0
MOVL C01671 V=800.0 PL=0
MOVL C01672 V=800.0 PL=0
MOVL C01673 V=800.0 PL=0
MOVL C01674 V=800.0 PL=0
MOVL C01675 V=800.0 PL=0
MOVL C01676 V=800.0 PL=0
MOVL C01677 V=800.0 PL=0
MOVL C01678 V=800.0 PL=0
MOVL C01679 V=800.0 PL=0
MOVL C01680 V=800.0 PL=0
MOVL C01681 V=800.0 PL=0
MOVL C01682 V=800.0 PL=0
MOVL C01683 V=800.0 PL=0
MOVL C01684 V=800.0 PL=0
MOVL C01685 V=800.0 PL=0
MOVL C01686 V=800.0 PL=0
MOVL C01687 V=800.0 PL=0
MOVL C01688 V=800.0 PL=0
MOVL C01689 V=800.0 PL=0
MOVL C01690 V=800.0 PL=0
MOVL C01691 V=800.0 PL=0
MOVL C01692 V=800.0 PL=0
MOVL C01693 V=800.0 PL=0
MOVL C01694 V=800.0 PL=0
MOVL C01695 V=800.0 PL=0
MOVL C01696 V=800.0 PL=0
MOVL C01697 V=800.0 PL=0
MOVL C01698 V=800.0 PL=0
MOVL C01699 V=800.0 PL=0
MOVL C01700 V=800.0 PL=0
MOVL C01701 V=800.0 PL=0
MOVL C01702 V=800.0 PL=0
MOVL C01703 V=800.0 PL=0
MOVL C01704 V=800.0 PL=0
MOVL C01705 V=800.0 PL=0
MOVL C01706 V=800.0 PL=0
MOVL C01707 V=800.0 PL=0
MOVL C01708 V=800.0 PL=0
MOVL C01709 V=800.0 PL=0
MOVL C01710 V=800.0 PL=0
MOVL C01711 V=800.0 PL=0
MOVL C01712 V=800.0 PL=0
MOVL C01713 V=800.0 PL=0
MOVL C01714 V=800.0 PL=0
MOVL C01715 V=800.0 PL=0
MOVL C01716 V=800.0 PL=0
MOVL C01717 V=800.0 PL=0
MOVL C01718 V=800.0 PL=0
MOVL C01719 V=800.0 PL=0
MOVL C01720 V=800.0 PL=0
MOVL C01721 V=800.0 PL=0
MOVL C01722 V=800.0 PL=0
MOVL C01723 V=800.0 PL=0
MOVL C01724 V=800.0 PL=0
MOVL C01725 V=800.0 PL=0
MOVL C01726 V=800.0 PL=0
MOVL C01727 V=800.0 PL=0
MOVL C01728 V=800.0 PL=0
MOVL C01729 V=800.0 PL=0
MOVL C01730 V=800.0 PL=0
MOVL C01731 V=800.0 PL=0
MOVL C01732 V=800.0 PL=0
MOVL C01733 V=800.0 PL=0
MOVL C01734 V=800.0 PL=0
MOVL C01735 V=800.0 PL=0
MOVL C01736 V=800.0 PL=0
MOVL C01737 V=800.0 PL=0
MOVL C01738 V=800.0 PL=0
MOVL C01739 V=800.0 PL=0
MOVL C01740 V=800.0 PL=0
MOVL C01741 V=800.0 PL=0
MOVL C01742 V=800.0 PL=0
MOVL C01743 V=800.0 PL=0
MOVL C01744 V=800.0 PL=0
MOVL C01745 V=800.0 PL=0
MOVL C01746 V=800.0 PL=0
MOVL C01747 V=800.0 PL=0
MOVL C01748 V=800.0 PL=0
MOVL C01749 V=800.0 PL=0
MOVL C01750 V=800.0 PL=0
MOVL C01751 V=800.0 PL=0
MOVL C01752 V=800.0 PL=0
MOVL C01753 V=800.0 PL=0
MOVL C01754 V=800.0 PL=0
MOVL C01755 V=800.0 PL=0
MOVL C01756 V=800.0 PL=0
MOVL C01757 V=800.0 PL=0
MOVL C01758 V=800.0 PL=0
MOVL C01759 V=800.0 PL=0
MOVL C01760 V=800.0 PL=0
MOVL C01761 V=800.0 PL=0
MOVL C01762 V=800.0 PL=0
MOVL C01763 V=800.0 PL=0
MOVL C01764 V=800.0 PL=0
MOVL C01765 V=800.0 PL=0
MOVL C01766 V=800.0 PL=0
MOVL C01767 V=800.0 PL=0
MOVL C01768 V=800.0 PL=0
MOVL C01769 V=800.0 PL=0
MOVL C01770 V=800.0 PL=0
MOVL C01771 V=800.0 PL=0
MOVL C01772 V=800.0 PL=0
MOVL C01773 V=800.0 PL=0
MOVL C01774 V=800.0 PL=0
MOVL C01775 V=800.0 PL=0
MOVL C01776 V=800.0 PL=0
MOVL C01777 V=800.0 PL=0
MOVL C01778 V=800.0 PL=0
MOVL C01779 V=800.0 PL=0
MOVL C01780 V=800.0 PL=0
MOVL C01781 V=800.0 PL=0
MOVL C01782 V=800.0 PL=0
MOVL C01783 V=800.0 PL=0
MOVL C01784 V=800.0 PL=0
MOVL C01785 V=800.0 PL=0
MOVL C01786 V=800.0 PL=0
MOVL C01787 V=800.0 PL=0
MOVL C01788 V=800.0 PL=0
MOVL C01789 V=800.0 PL=0
MOVL C01790 V=800.0 PL=0
MOVL C01791 V=800.0 PL=0
MOVL C01792 V=800.0 PL=0
MOVL C01793 V=800.0 PL=0
MOVL C01794 V=800.0 PL=0
MOVL C01795 V=800.0 PL=0
MOVL C01796 V=800.0 PL=0
MOVL C01797 V=800.0 PL=0
MOVL C01798 V=800.0 PL=0
MOVL C01799 V=800.0 PL=0
MOVL C01800 V=800.0 PL=0
MOVL C01801 V=800.0 PL=0
MOVL C01802 V=800.0 PL=0
MOVL C01803 V=800.0 PL=0
MOVL C01804 V=800.0 PL=0
MOVL C01805 V=800.0 PL=0
MOVL C01806 V=800.0 PL=0
MOVL C01807 V=800.0 PL=0
MOVL C01808 V=800.0 PL=0
MOVL C01809 V=800.0 PL=0
MOVL C01810 V=800.0 PL=0
MOVL C01811 V=800.0 PL=0
MOVL C01812 V=800.0 PL=0
MOVL C01813 V=800.0 PL=0
MOVL C01814 V=800.0 PL=0
MOVL C01815 V=800.0 PL=0
MOVL C01816 V=800.0 PL=0
MOVL C01817 V=800.0 PL=0
MOVL C01818 V=800.0 PL=0
MOVL C01819 V=800.0 PL=0
MOVL C01820 V=800.0 PL=0
MOVL C01821 V=800.0 PL=0
MOVL C01822 V=800.0 PL=0
MOVL C01823 V=800.0 PL=0
MOVL C01824 V=800.0 PL=0
MOVL C01825 V=800.0 PL=0
MOVL C01826 V=800.0 PL=0
MOVL C01827 V=800.0 PL=0
MOVL C01828 V=800.0 PL=0
MOVL C01829 V=800.0 PL=0
MOVL C01830 V=800.0 PL=0
MOVL C01831 V=800.0 PL=0
MOVL C01832 V=800.0 PL=0
MOVL C01833 V=800.0 PL=0
MOVL C01834 V=800.0 PL=0
MOVL C01835 V=800.0 PL=0
MOVL C01836 V=800.0 PL=0
MOVL C01837 V=800.0 PL=0
MOVL C01838 V=800.0 PL=0
MOVL C01839 V=800.0 PL=0
MOVL C01840 V=800.0 PL=0
MOVL C01841 V=800.0 PL=0
MOVL C01842 V=800.0 PL=0
MOVL C01843 V=800.0 PL=0
MOVL C01844 V=800.0 PL=0
MOVL C01845 V=800.0 PL=0
MOVL C01846 V=800.0 PL=0
MOVL C01847 V=800.0 PL=0
MOVL C01848 V=800.0 PL=0
MOVL C01849 V=800.0 PL=0
MOVL C01850 V=800.0 PL=0
MOVL C01851 V=800.0 PL=0
MOVL C01852 V=800.0 PL=0
MOVL C01853 V=800.0 PL=0
MOVL C01854 V=800.0 PL=0
MOVL C01855 V=800.0 PL=0
MOVL C01856 V=800.0 PL=0
MOVL C01857 V=800.0 PL=0
MOVL C01858 V=800.0 PL=0
MOVL C01859 V=800.0 PL=0
MOVL C01860 V=800.0 PL=0
MOVL C01861 V=800.0 PL=0
MOVL C01862 V=800.0 PL=0
MOVL C01863 V=800.0 PL=0
MOVL C01864 V=800.0 PL=0
MOVL C01865 V=800.0 PL=0
MOVL C01866 V=800.0 PL=0
MOVL C01867 V=800.0 PL=0
MOVL C01868 V=800.0 PL=0
MOVL C01869 V=800.0 PL=0
MOVL C01870 V=800.0 PL=0
MOVL C01871 V=800.0 PL=0
MOVL C01872 V=800.0 PL=0
MOVL C01873 V=800.0 PL=0
MOVL C01874 V=800.0 PL=0
MOVL C01875 V=800.0 PL=0
MOVL C01876 V=800.0 PL=0
MOVL C01877 V=800.0 PL=0
MOVL C01878 V=800.0 PL=0
MOVL C01879 V=800.0 PL=0
MOVL C01880 V=800.0 PL=0
MOVL C01881 V=800.0 PL=0
MOVL C01882 V=800.0 PL=0
MOVL C01883 V=800.0 PL=0
MOVL C01884 V=800.0 PL=0
MOVL C01885 V=800.0 PL=0
MOVL C01886 V=800.0 PL=0
MOVL C01887 V=800.0 PL=0
MOVL C01888 V=800.0 PL=0
MOVL C01889 V=800.0 PL=0
MOVL C01890 V=800.0 PL=0
MOVL C01891 V=800.0 PL=0
MOVL C01892 V=800.0 PL=0
MOVL C01893 V=800.0 PL=0
MOVL C01894 V=800.0 PL=0
MOVL C01895 V=800.0 PL=0
MOVL C01896 V=800.0 PL=0
MOVL C01897 V=800.0 PL=0
MOVL C01898 V=800.0 PL=0
MOVL C01899 V=800.0 PL=0
MOVL C01900 V=800.0 PL=0
MOVL C01901 V=800.0 PL=0
MOVL C01902 V=800.0 PL=0
MOVL C01903 V=800.0 PL=0
MOVL C01904 V=800.0 PL=0
MOVL C01905 V=800.0 PL=0
MOVL C01906 V=800.0 PL=0
MOVL C01907 V=800.0 PL=0
MOVL C01908 V=800.0 PL=0
MOVL C01909 V=800.0 PL=0
MOVL C01910 V=800.0 PL=0
MOVL C01911 V=800.0 PL=0
MOVL C01912 V=800.0 PL=0
MOVL C01913 V=800.0 PL=0
MOVL C01914 V=800.0 PL=0
MOVL C01915 V=800.0 PL=0
MOVL C01916 V=800.0 PL=0
MOVL C01917 V=800.0 PL=0
MOVL C01918 V=800.0 PL=0
MOVL C01919 V=800.0 PL=0
MOVL C01920 V=800.0 PL=0
MOVL C01921 V=800.0 PL=0
MOVL C01922 V=800.0 PL=0
MOVL C01923 V=800.0 PL=0
MOVL C01924 V=800.0 PL=0
MOVL C01925 V=800.0 PL=0
MOVL C01926 V=800.0 PL=0
MOVL C01927 V=800.0 PL=0
MOVL C01928 V=800.0 PL=0
MOVL C01929 V=800.0 PL=0
MOVL C01930 V=800.0 PL=0
MOVL C01931 V=800.0 PL=0
MOVL C01932 V=800.0 PL=0
MOVL C01933 V=800.0 PL=0
MOVL C01934 V=800.0 PL=0
MOVL C01935 V=800.0 PL=0
MOVL C01936 V=800.0 PL=0
MOVL C01937 V=800.0 PL=0
MOVL C01938 V=800.0 PL=0
MOVL C01939 V=800.0 PL=0
MOVL C01940 V=800.0 PL=0
MOVL C01941 V=800.0 PL=0
MOVL C01942 V=800.0 PL=0
MOVL C01943 V=800.0 PL=0
MOVL C01944 V=800.0 PL=0
MOVL C01945 V=800.0 PL=0
MOVL C01946 V=800.0 PL=0
MOVL C01947 V=800.0 PL=0
MOVL C01948 V=800.0 PL=0
MOVL C01949 V=800.0 PL=0
MOVL C01950 V=800.0 PL=0
MOVL C01951 V=800.0 PL=0
MOVL C01952 V=800.0 PL=0
MOVL C01953 V=800.0 PL=0
MOVL C01954 V=800.0 PL=0
MOVL C01955 V=800.0 PL=0
MOVL C01956 V=800.0 PL=0
MOVL C01957 V=800.0 PL=0
MOVL C01958 V=800.0 PL=0
MOVL C01959 V=800.0 PL=0
MOVL C01960 V=800.0 PL=0
MOVL C01961 V=800.0 PL=0
MOVL C01962 V=800.0 PL=0
MOVL C01963 V=800.0 PL=0
MOVL C01964 V=800.0 PL=0
MOVL C01965 V=800.0 PL=0
MOVL C01966 V=800.0 PL=0
MOVL C01967 V=800.0 PL=0
MOVL C01968 V=800.0 PL=0
MOVL C01969 V=800.0 PL=0
MOVL C01970 V=800.0 PL=0
MOVL C01971 V=800.0 PL=0
MOVL C01972 V=800.0 PL=0
MOVL C01973 V=800.0 PL=0
MOVL C01974 V=800.0 PL=0
MOVL C01975 V=800.0 PL=0
MOVL C01976 V=800.0 PL=0
MOVL C01977 V=800.0 PL=0
MOVL C01978 V=800.0 PL=0
MOVL C01979 V=800.0 PL=0
MOVL C01980 V=800.0 PL=0
MOVL C01981 V=800.0 PL=0
MOVL C01982 V=800.0 PL=0
MOVL C01983 V=800.0 PL=0
MOVL C01984 V=800.0 PL=0
MOVL C01985 V=800.0 PL=0
MOVL C01986 V=800.0 PL=0
MOVL C01987 V=800.0 PL=0
MOVL C01988 V=800.0 PL=0
MOVL C01989 V=800.0 PL=0
MOVL C01990 V=800.0 PL=0
MOVL C01991 V=800.0 PL=0
MOVL C01992 V=800.0 PL=0
MOVL C01993 V=800.0 PL=0
MOVL C01994 V=800.0 PL=0
MOVL C01995 V=800.0 PL=0
MOVL C01996 V=800.0 PL=0
MOVL C01997 V=800.0 PL=0
MOVL C01998 V=800.0 PL=0
MOVL C01999 V=800.0 PL=0
MOVL C02000 V=800.0 PL=0
MOVL C02001 V=800.0 PL=0
MOVL C02002 V=800.0 PL=0
MOVL C02003 V=800.0 PL=0
MOVL C02004 V=800.0 PL=0
MOVL C02005 V=800.0 PL=0
MOVL C02006 V=800.0 PL=0
MOVL C02007 V=800.0 PL=0
MOVL C02008 V=800.0 PL=0
MOVL C02009 V=800.0 PL=0
MOVL C02010 V=800.0 PL=0
MOVL C02011 V=800.0 PL=0
MOVL C02012 V=800.0 PL=0
MOVL C02013 V=800.0 PL=0
MOVL C02014 V=800.0 PL=0
MOVL C02015 V=800.0 PL=0
MOVL C02016 V=800.0 PL=0
MOVL C02017 V=800.0 PL=0
MOVL C02018 V=800.0 PL=0
MOVL C02019 V=800.0 PL=0
MOVL C02020 V=800.0 PL=0
MOVL C02021 V=800.0 PL=0
MOVL C02022 V=800.0 PL=0
MOVL C02023 V=800.0 PL=0
MOVL C02024 V=800.0 PL=0
MOVL C02025 V=800.0 PL=0
MOVL C02026 V=800.0 PL=0
MOVL C02027 V=800.0 PL=0
MOVL C02028 V=800.0 PL=0
MOVL C02029 V=800.0 PL=0
MOVL C02030 V=800.0 PL=0
MOVL C02031 V=800.0 PL=0
MOVL C02032 V=800.0 PL=0
MOVL C02033 V=800.0 PL=0
MOVL C02034 V=800.0 PL=0
MOVL C02035 V=800.0 PL=0
MOVL C02036 V=800.0 PL=0
MOVL C02037 V=800.0 PL=0
MOVL C02038 V=800.0 PL=0
MOVL C02039 V=800.0 PL=0
MOVL C02040 V=800.0 PL=0
MOVL C02041 V=800.0 PL=0
MOVL C02042 V=800.0 PL=0
MOVL C02043 V=800.0 PL=0
MOVL C02044 V=800.0 PL=0
MOVL C02045 V=800.0 PL=0
MOVL C02046 V=800.0 PL=0
MOVL C02047 V=800.0 PL=0
MOVL C02048 V=800.0 PL=0
MOVL C02049 V=800.0 PL=0
MOVL C02050 V=800.0 PL=0
MOVL C02051 V=800.0 PL=0
MOVL C02052 V=800.0 PL=0
MOVL C02053 V=800.0 PL=0
MOVL C02054 V=800.0 PL=0
MOVL C02055 V=800.0 PL=0
MOVL C02056 V=800.0 PL=0
MOVL C02057 V=800.0 PL=0
MOVL C02058 V=800.0 PL=0
MOVL C02059 V=800.0 PL=0
MOVL C02060 V=800.0 PL=0
MOVL C02061 V=800.0 PL=0
MOVL C02062 V=800.0 PL=0
MOVL C02063 V=800.0 PL=0
MOVL C02064 V=800.0 PL=0
MOVL C02065 V=800.0 PL=0
MOVL C02066 V=800.0 PL=0
MOVL C02067 V=800.0 PL=0
MOVL C02068 V=800.0 PL=0
MOVL C02069 V=800.0 PL=0
MOVL C02070 V=800.0 PL=0
MOVL C02071 V=800.0 PL=0
MOVL C02072 V=800.0 PL=0
MOVL C02073 V=800.0 PL=0
MOVL C02074 V=800.0 PL=0
MOVL C02075 V=800.0 PL=0
MOVL C02076 V=800.0 PL=0
MOVL C02077 V=800.0 PL=0
MOVL C02078 V=800.0 PL=0
MOVL C02079 V=800.0 PL=0
MOVL C02080 V=800.0 PL=0
MOVL C02081 V=800.0 PL=0
MOVL C02082 V=800.0 PL=0
MOVL C02083 V=800.0 PL=0
MOVL C02084 V=800.0 PL=0
MOVL C02085 V=800.0 PL=0
MOVL C02086 V=800.0 PL=0
MOVL C02087 V=800.0 PL=0
MOVL C02088 V=800.0 PL=0
MOVL C02089 V=800.0 PL=0
MOVL C02090 V=800.0 PL=0
MOVL C02091 V=800.0 PL=0
MOVL C02092 V=800.0 PL=0
MOVL C02093 V=800.0 PL=0
MOVL C02094 V=800.0 PL=0
MOVL C02095 V=800.0 PL=0
MOVL C02096 V=800.0 PL=0
MOVL C02097 V=800.0 PL=0
MOVL C02098 V=800.0 PL=0
MOVL C02099 V=800.0 PL=0
MOVL C02100 V=800.0 PL=0
MOVL C02101 V=800.0 PL=0
MOVL C02102 V=800.0 PL=0
MOVL C02103 V=800.0 PL=0
MOVL C02104 V=800.0 PL=0
MOVL C02105 V=800.0 PL=0
MOVL C02106 V=800.0 PL=0
MOVL C02107 V=800.0 PL=0
MOVL C02108 V=800.0 PL=0
MOVL C02109 V=800.0 PL=0
MOVL C02110 V=800.0 PL=0
MOVL C02111 V=800.0 PL=0
MOVL C02112 V=800.0 PL=0
MOVL C02113 V=800.0 PL=0
MOVL C02114 V=800.0 PL=0
MOVL C02115 V=800.0 PL=0
MOVL C02116 V=800.0 PL=0
MOVL C02117 V=800.0 PL=0
MOVL C02118 V=800.0 PL=0
MOVL C02119 V=800.0 PL=0
MOVL C02120 V=800.0 PL=0
MOVL C02121 V=800.0 PL=0
MOVL C02122 V=800.0 PL=0
MOVL C02123 V=800.0 PL=0
MOVL C02124 V=800.0 PL=0
MOVL C02125 V=800.0 PL=0
MOVL C02126 V=800.0 PL=0
MOVL C02127 V=800.0 PL=0
MOVL C02128 V=800.0 PL=0
MOVL C02129 V=800.0 PL=0
MOVL C02130 V=800.0 PL=0
MOVL C02131 V=800.0 PL=0
MOVL C02132 V=800.0 PL=0
MOVL C02133 V=800.0 PL=0
MOVL C02134 V=800.0 PL=0
MOVL C02135 V=800.0 PL=0
MOVL C02136 V=800.0 PL=0
MOVL C02137 V=800.0 PL=0
MOVL C02138 V=800.0 PL=0
MOVL C02139 V=800.0 PL=0
MOVL C02140 V=800.0 PL=0
MOVL C02141 V=800.0 PL=0
MOVL C02142 V=800.0 PL=0
MOVL C02143 V=800.0 PL=0
MOVL C02144 V=800.0 PL=0
MOVL C02145 V=800.0 PL=0
MOVL C02146 V=800.0 PL=0
MOVL C02147 V=800.0 PL=0
MOVL C02148 V=800.0 PL=0
MOVL C02149 V=800.0 PL=0
MOVL C02150 V=800.0 PL=0
MOVL C02151 V=800.0 PL=0
MOVL C02152 V=800.0 PL=0
MOVL C02153 V=800.0 PL=0
MOVL C02154 V=800.0 PL=0
MOVL C02155 V=800.0 PL=0
MOVL C02156 V=800.0 PL=0
MOVL C02157 V=800.0 PL=0
MOVL C02158 V=800.0 PL=0
MOVL C02159 V=800.0 PL=0
MOVL C02160 V=800.0 PL=0
MOVL C02161 V=800.0 PL=0
MOVL C02162 V=800.0 PL=0
MOVL C02163 V=800.0 PL=0
MOVL C02164 V=800.0 PL=0
MOVL C02165 V=800.0 PL=0
